REGION Network 4
   RUNG wire#powerrail
      Contact( #Start )
      S_SR(operand := #Automat, r1 := wire#w1)
      S_OFFDT(T_NO := "Spoždění ukončení automatu", TV := S5T#4s, R :=, BI =>, RET_VAL =>)
      Coil( #"Automat Delay" )
   END_RUNG
   RUNG wire#powerrail
      Contact( #Stop )
   END_RUNG wire#w1
   RUNG wire#powerrail
      Contact( "OPPovely"."OP Manual" )
   END_RUNG wire#w1
   // the same network as SCL:
   IF #Start THEN
       #Automat := TRUE;   // SR flip-flop
   END_IF;
   IF #Stop OR "OPPovely"."OP Manual" THEN #Automat := FALSE; END_IF;
   #_s5time1 := S_OFFDT(T_NO := "Spoždění ukončení automatu", S := #Automat, TV := S5T#4s, Q => #_w1);
   #"Automat Delay" := #_w1;
END_REGION

REGION Network 5
   RUNG wire#powerrail
      #"Vyhodnocení hran_Instance"(input := %DB20.DBD0, positive => %DB21.DBD0, negative => %DB22.DBD0)
   END_RUNG
   // the same network as SCL:
   #"Vyhodnocení hran_Instance"(input := %DB20.DBD0, positive => %DB21.DBD0, negative => %DB22.DBD0);   // "Vyhodnocení hran"
END_REGION

REGION Network 6
   RUNG wire#powerrail
      #"Vyhodnocení hran_Instance_Linka 1"(input := %DB20.DBD4, positive => %DB21.DBD4, negative => %DB22.DBD4)
   END_RUNG
   // the same network as SCL:
   #"Vyhodnocení hran_Instance_Linka 1"(input := %DB20.DBD4, positive => %DB21.DBD4, negative => %DB22.DBD4);   // "Vyhodnocení hran"
END_REGION

REGION Network 7
   RUNG wire#powerrail
      Contact( "Tag_64" )
      Coil( "Tag_65" )
   END_RUNG
   // the same network as SCL:
   "Tag_65" := "Tag_64";
END_REGION
END_FUNCTION_BLOCK

FUNCTION_BLOCK "Dopravníky palet_2"   // FB7, LAD
{ S7_Optimized_Access := 'FALSE' }
VERSION : 0.1
   VAR
      Přesun : Struct
         KonecD4naDestohovač : Bool;
         DestohovačNaKonecD5 : Bool;
         KonecD5naZačátekD8 : Bool;
         ZačátekD8naD8pozice12 : Bool;
         D8pozice12naD8pozice11 : Bool;
         D8pozice12naD12 : Bool;
         D8pozice11naD11 : Bool;
         D12naD17pozice12 : Bool;
         D11naD17pozice11 : Bool;
         D17pozice12naKonecP17 : Bool;
         D17pozice11naKonecP17 : Bool;
         KonecP17naZačátekP18 : Bool;
         ZačátekP18naKonecP18 : Bool;
         KonecP18naP19 : Bool;
         P19naZačátekP20 : Bool;
         ZačátekP20naKonecP20 : Bool;
         KonecP20NaP21 : Bool;
      END_STRUCT;
      "Přítomnosti palet" : Struct
         PaletaPodDestohovačem : Bool;
         PaletaNaKonciD5 : Bool;
         PaletaNaZačátkuD8 : Bool;
         PaletaNaD8pozice12 : Bool;
         PaletaNaD8pozice11 : Bool;
         PaletaNaP12 : Bool;
         PaletaNaP11 : Bool;
         PaletaNaD17pozice12 : Bool;
         PaletaNaD17pozice11 : Bool;
         PaletaNaKonciP17 : Bool;
         "PaletaNaZačátku P18" : Bool;
         PaletaNaKonciP18 : Bool;
         PaletaNaP19 : Bool;
         PaletaNaZačátkuP20 : Bool;
         PaletaNaKonciP20 : Bool;
      END_STRUCT;
      "Nájezdy palet" : Struct
         PaletaPodDestohovačem : Bool;
         PaletaNaKonciD5 : Bool;
         PaletaNaZačátkuD8 : Bool;
         PaletaNaD8pozice12 : Bool;
         PaletaNaD8pozice11 : Bool;
         PaletaNaP12 : Bool;
         PaletaNaP11 : Bool;
         PaletaNaD17pozice12 : Bool;
         PaletaNaD17pozice11 : Bool;
         PaletaNaKonciP17 : Bool;
         "PaletaNaZačátku P18" : Bool;
         PaletaNaKonciP18 : Bool;
         PaletaNaP19 : Bool;
         PaletaNaZačátkuP20 : Bool;
         PaletaNaKonciP20 : Bool;
      END_STRUCT;
      Palety : Struct
         P12 : "Paleta";
         P11 : "Paleta";
         P17poziceP11 : "Paleta";
         P17poziceP12 : "Paleta";
         KonecP17 : "Paleta";
         ZačátekP18 : "Paleta";
         KonecP18 : "Paleta";
         P19 : "Paleta";
         ZačátekP20 : "Paleta";
      END_STRUCT;
      Hrany : Struct
         T51Negativní : Bool;
      END_STRUCT;
      "Pallet dispenser_Instance" : "Pallet dispenser";
      "Přítomnost palety_Instance" : "Přítomnost palety";
   END_VAR
   VAR_TEMP
      Dummy : Bool;
      "Rovnání P11 sevřít" : Bool;
      "Rovnání P11 rozevřít" : Bool;
      "Rovnání P12 sevřít" : Bool;
      "Rovnání P12 rozevřít" : Bool;
      "Destohovač sevřít" : Bool;
      "Destohovač rozevřít" : Bool;
   END_VAR
   VAR_TEMP   // added for the SCL form of the ladder/FBD networks
      _s5time1 : S5Time;
      _w1 : Bool;
      _w2 : Bool;
      _w3 : Bool;
   END_VAR
BEGIN

REGION Network 1
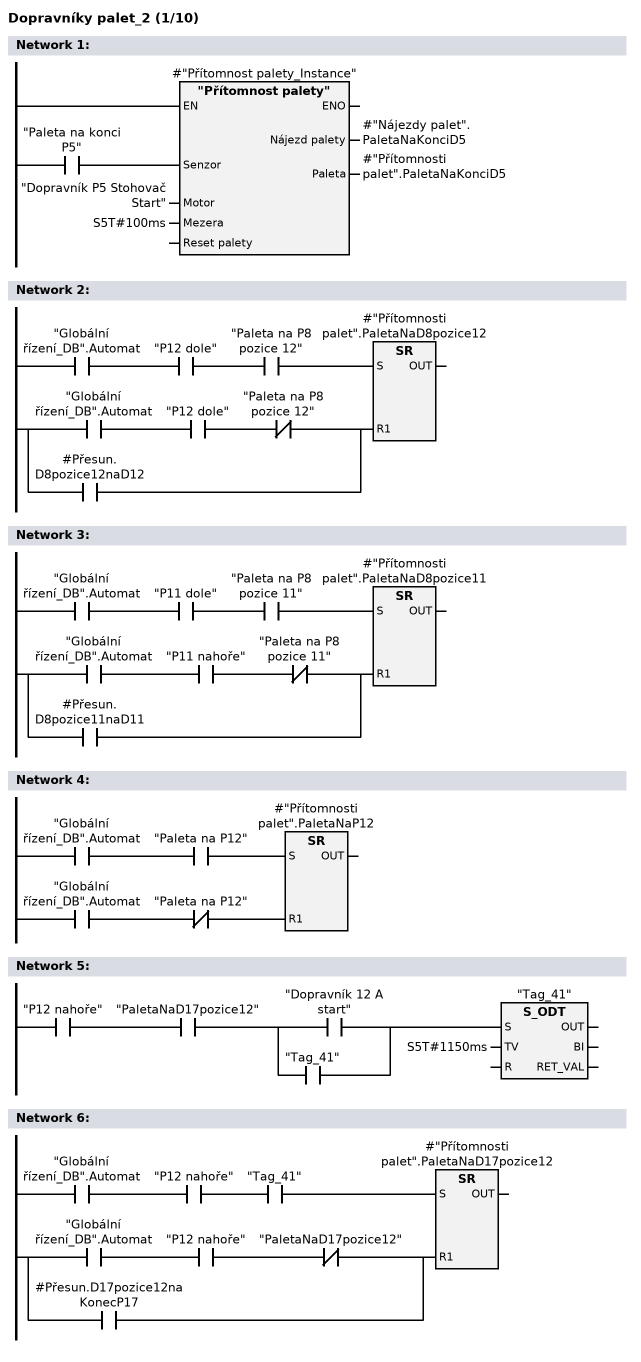
   RUNG wire#powerrail
      #"Přítomnost palety_Instance"(Senzor := wire#w1, Motor := "Dopravník P5 Stohovač Start", Mezera := S5T#100ms, "Reset palety" :=, "Nájezd palety" => #"Nájezdy palet".PaletaNaKonciD5, Paleta => #"Přítomnosti palet".PaletaNaKonciD5)
   END_RUNG
   RUNG wire#powerrail
      Contact( "Paleta na konci P5" )
   END_RUNG wire#w1
   // the same network as SCL:
   #"Přítomnost palety_Instance"(Senzor := "Paleta na konci P5",   // "Přítomnost palety"
                           Motor := "Dopravník P5 Stohovač Start",
                           Mezera := S5T#100ms,
                           "Nájezd palety" => #"Nájezdy palet".PaletaNaKonciD5,
                           Paleta => #"Přítomnosti palet".PaletaNaKonciD5);
END_REGION

REGION Network 2
   RUNG wire#powerrail
      Contact( "Globální řízení_DB".Automat )
      Contact( "P12 dole" )
      Contact( "Paleta na P8 pozice 12" )
      S_SR(operand := #"Přítomnosti palet".PaletaNaD8pozice12, r1 := wire#w1)
   END_RUNG
   RUNG wire#powerrail
      Contact( "Globální řízení_DB".Automat )
      Contact( "P12 dole" )
      I_Contact( "Paleta na P8 pozice 12" )
   END_RUNG wire#w1
   RUNG wire#powerrail
      Contact( #Přesun.D8pozice12naD12 )
   END_RUNG wire#w1
   // the same network as SCL:
   IF "Globální řízení_DB".Automat AND "P12 dole" AND "Paleta na P8 pozice 12" THEN
       #"Přítomnosti palet".PaletaNaD8pozice12 := TRUE;   // SR flip-flop
   END_IF;
   IF ("Globální řízení_DB".Automat AND "P12 dole" AND NOT "Paleta na P8 pozice 12") OR #Přesun.D8pozice12naD12 THEN
       #"Přítomnosti palet".PaletaNaD8pozice12 := FALSE;
   END_IF;
END_REGION

REGION Network 3
   RUNG wire#powerrail
      Contact( "Globální řízení_DB".Automat )
      Contact( "P11 dole" )
      Contact( "Paleta na P8 pozice 11" )
      S_SR(operand := #"Přítomnosti palet".PaletaNaD8pozice11, r1 := wire#w1)
   END_RUNG
   RUNG wire#powerrail
      Contact( "Globální řízení_DB".Automat )
      Contact( "P11 nahoře" )
      I_Contact( "Paleta na P8 pozice 11" )
   END_RUNG wire#w1
   RUNG wire#powerrail
      Contact( #Přesun.D8pozice11naD11 )
   END_RUNG wire#w1
   // the same network as SCL:
   IF "Globální řízení_DB".Automat AND "P11 dole" AND "Paleta na P8 pozice 11" THEN
       #"Přítomnosti palet".PaletaNaD8pozice11 := TRUE;   // SR flip-flop
   END_IF;
   IF ("Globální řízení_DB".Automat AND "P11 nahoře" AND NOT "Paleta na P8 pozice 11") OR #Přesun.D8pozice11naD11 THEN
       #"Přítomnosti palet".PaletaNaD8pozice11 := FALSE;
   END_IF;
END_REGION

REGION Network 4
   RUNG wire#powerrail
      Contact( "Globální řízení_DB".Automat )
      Contact( "Paleta na P12" )
      S_SR(operand := #"Přítomnosti palet".PaletaNaP12, r1 := wire#w1)
   END_RUNG
   RUNG wire#powerrail
      Contact( "Globální řízení_DB".Automat )
      I_Contact( "Paleta na P12" )
   END_RUNG wire#w1
   // the same network as SCL:
   IF "Globální řízení_DB".Automat AND "Paleta na P12" THEN
       #"Přítomnosti palet".PaletaNaP12 := TRUE;   // SR flip-flop
   END_IF;
   IF "Globální řízení_DB".Automat AND NOT "Paleta na P12" THEN
       #"Přítomnosti palet".PaletaNaP12 := FALSE;
   END_IF;
END_REGION

REGION Network 5
   RUNG wire#powerrail
      Contact( "P12 nahoře" )
      Contact( "PaletaNaD17pozice12" )
      wire#w1
      Contact( "Dopravník 12 A start" )
      wire#w2
      S_ODT(T_NO := "Tag_41", TV := S5T#1150ms, R :=, BI =>, RET_VAL =>)
   END_RUNG
   RUNG wire#w1
      Contact( "Tag_41" )
   END_RUNG wire#w2
   // the same network as SCL:
   #_s5time1 := S_ODT(T_NO := "Tag_41",
                      S := "P12 nahoře" AND "PaletaNaD17pozice12" AND ("Dopravník 12 A start" OR "Tag_41"),
                      TV := S5T#1150ms);
END_REGION

REGION Network 6
   RUNG wire#powerrail
      Contact( "Globální řízení_DB".Automat )
      Contact( "P12 nahoře" )
      Contact( "Tag_41" )
      S_SR(operand := #"Přítomnosti palet".PaletaNaD17pozice12, r1 := wire#w1)
   END_RUNG
   RUNG wire#powerrail
      Contact( "Globální řízení_DB".Automat )
      Contact( "P12 nahoře" )
      I_Contact( "PaletaNaD17pozice12" )
   END_RUNG wire#w1
   RUNG wire#powerrail
      Contact( #Přesun.D17pozice12naKonecP17 )
   END_RUNG wire#w1
   // the same network as SCL:
   IF "Globální řízení_DB".Automat AND "P12 nahoře" AND "Tag_41" THEN
       #"Přítomnosti palet".PaletaNaD17pozice12 := TRUE;   // SR flip-flop
   END_IF;
   IF ("Globální řízení_DB".Automat AND "P12 nahoře" AND NOT "PaletaNaD17pozice12") OR #Přesun.D17pozice12naKonecP17 THEN
       #"Přítomnosti palet".PaletaNaD17pozice12 := FALSE;
   END_IF;
END_REGION

REGION Network 7
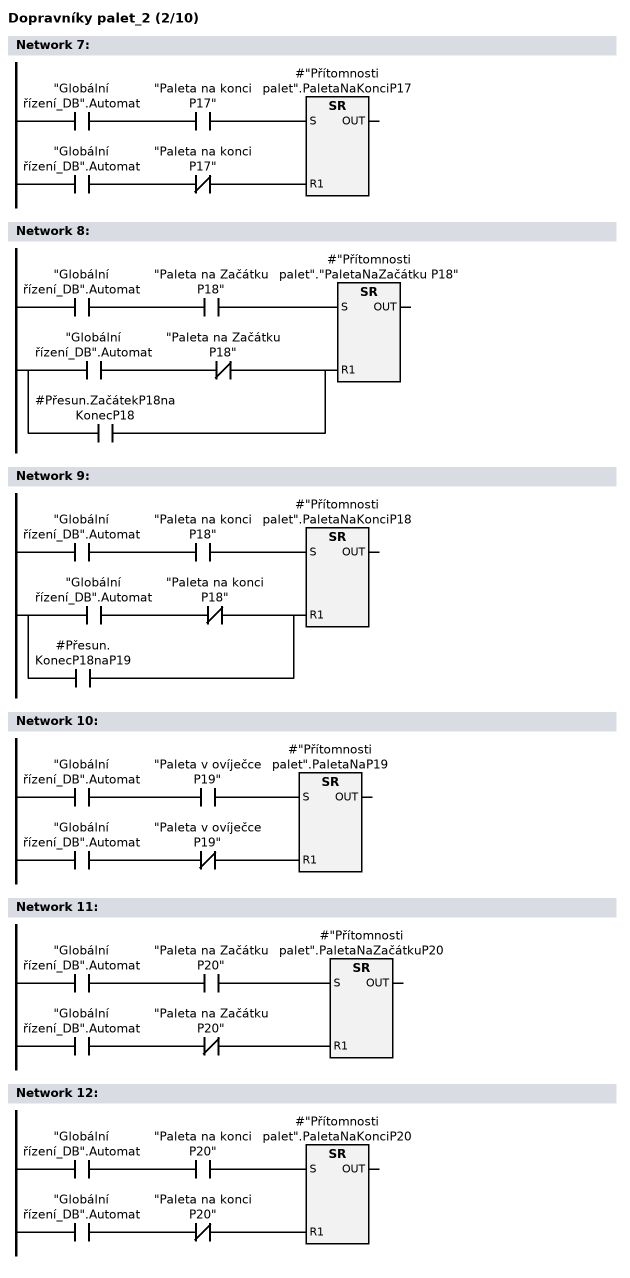
   RUNG wire#powerrail
      Contact( "Globální řízení_DB".Automat )
      Contact( "Paleta na konci P17" )
      S_SR(operand := #"Přítomnosti palet".PaletaNaKonciP17, r1 := wire#w1)
   END_RUNG
   RUNG wire#powerrail
      Contact( "Globální řízení_DB".Automat )
      I_Contact( "Paleta na konci P17" )
   END_RUNG wire#w1
   // the same network as SCL:
   IF "Globální řízení_DB".Automat AND "Paleta na konci P17" THEN
       #"Přítomnosti palet".PaletaNaKonciP17 := TRUE;   // SR flip-flop
   END_IF;
   IF "Globální řízení_DB".Automat AND NOT "Paleta na konci P17" THEN
       #"Přítomnosti palet".PaletaNaKonciP17 := FALSE;
   END_IF;
END_REGION

REGION Network 8
   RUNG wire#powerrail
      Contact( "Globální řízení_DB".Automat )
      Contact( "Paleta na Začátku P18" )
      S_SR(operand := #"Přítomnosti palet"."PaletaNaZačátku P18", r1 := wire#w1)
   END_RUNG
   RUNG wire#powerrail
      Contact( "Globální řízení_DB".Automat )
      I_Contact( "Paleta na Začátku P18" )
   END_RUNG wire#w1
   RUNG wire#powerrail
      Contact( #Přesun.ZačátekP18naKonecP18 )
   END_RUNG wire#w1
   // the same network as SCL:
   IF "Globální řízení_DB".Automat AND "Paleta na Začátku P18" THEN
       #"Přítomnosti palet"."PaletaNaZačátku P18" := TRUE;   // SR flip-flop
   END_IF;
   IF ("Globální řízení_DB".Automat AND NOT "Paleta na Začátku P18") OR #Přesun.ZačátekP18naKonecP18 THEN
       #"Přítomnosti palet"."PaletaNaZačátku P18" := FALSE;
   END_IF;
END_REGION

REGION Network 9
   RUNG wire#powerrail
      Contact( "Globální řízení_DB".Automat )
      Contact( "Paleta na konci P18" )
      S_SR(operand := #"Přítomnosti palet".PaletaNaKonciP18, r1 := wire#w1)
   END_RUNG
   RUNG wire#powerrail
      Contact( "Globální řízení_DB".Automat )
      I_Contact( "Paleta na konci P18" )
   END_RUNG wire#w1
   RUNG wire#powerrail
      Contact( #Přesun.KonecP18naP19 )
   END_RUNG wire#w1
   // the same network as SCL:
   IF "Globální řízení_DB".Automat AND "Paleta na konci P18" THEN
       #"Přítomnosti palet".PaletaNaKonciP18 := TRUE;   // SR flip-flop
   END_IF;
   IF ("Globální řízení_DB".Automat AND NOT "Paleta na konci P18") OR #Přesun.KonecP18naP19 THEN
       #"Přítomnosti palet".PaletaNaKonciP18 := FALSE;
   END_IF;
END_REGION

REGION Network 10
   RUNG wire#powerrail
      Contact( "Globální řízení_DB".Automat )
      Contact( "Paleta v ovíječce P19" )
      S_SR(operand := #"Přítomnosti palet".PaletaNaP19, r1 := wire#w1)
   END_RUNG
   RUNG wire#powerrail
      Contact( "Globální řízení_DB".Automat )
      I_Contact( "Paleta v ovíječce P19" )
   END_RUNG wire#w1
   // the same network as SCL:
   IF "Globální řízení_DB".Automat AND "Paleta v ovíječce P19" THEN
       #"Přítomnosti palet".PaletaNaP19 := TRUE;   // SR flip-flop
   END_IF;
   IF "Globální řízení_DB".Automat AND NOT "Paleta v ovíječce P19" THEN
       #"Přítomnosti palet".PaletaNaP19 := FALSE;
   END_IF;
END_REGION

REGION Network 11
   RUNG wire#powerrail
      Contact( "Globální řízení_DB".Automat )
      Contact( "Paleta na Začátku P20" )
      S_SR(operand := #"Přítomnosti palet".PaletaNaZačátkuP20, r1 := wire#w1)
   END_RUNG
   RUNG wire#powerrail
      Contact( "Globální řízení_DB".Automat )
      I_Contact( "Paleta na Začátku P20" )
   END_RUNG wire#w1
   // the same network as SCL:
   IF "Globální řízení_DB".Automat AND "Paleta na Začátku P20" THEN
       #"Přítomnosti palet".PaletaNaZačátkuP20 := TRUE;   // SR flip-flop
   END_IF;
   IF "Globální řízení_DB".Automat AND NOT "Paleta na Začátku P20" THEN
       #"Přítomnosti palet".PaletaNaZačátkuP20 := FALSE;
   END_IF;
END_REGION

REGION Network 12
   RUNG wire#powerrail
      Contact( "Globální řízení_DB".Automat )
      Contact( "Paleta na konci P20" )
      S_SR(operand := #"Přítomnosti palet".PaletaNaKonciP20, r1 := wire#w1)
   END_RUNG
   RUNG wire#powerrail
      Contact( "Globální řízení_DB".Automat )
      I_Contact( "Paleta na konci P20" )
   END_RUNG wire#w1
   // the same network as SCL:
   IF "Globální řízení_DB".Automat AND "Paleta na konci P20" THEN
       #"Přítomnosti palet".PaletaNaKonciP20 := TRUE;   // SR flip-flop
   END_IF;
   IF "Globální řízení_DB".Automat AND NOT "Paleta na konci P20" THEN
       #"Přítomnosti palet".PaletaNaKonciP20 := FALSE;
   END_IF;
END_REGION

REGION Network 13
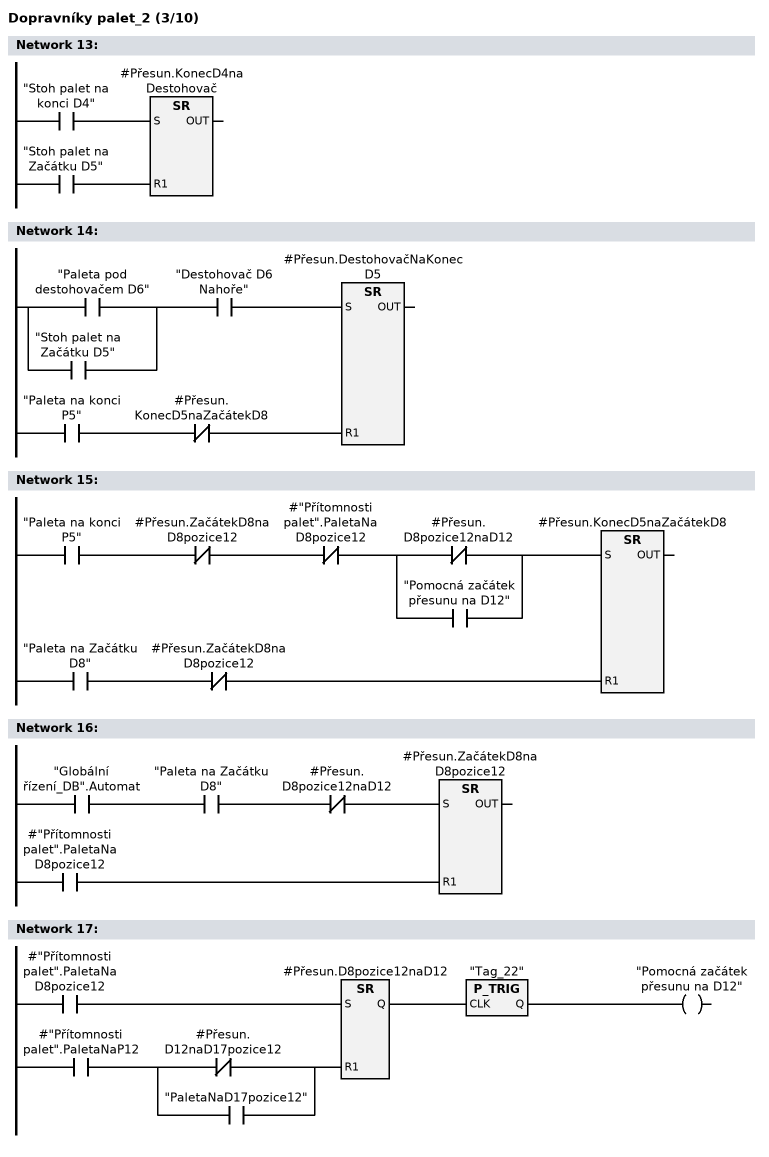
   RUNG wire#powerrail
      Contact( "Stoh palet na konci D4" )
      S_SR(operand := #Přesun.KonecD4naDestohovač, r1 := wire#w1)
   END_RUNG
   RUNG wire#powerrail
      Contact( "Stoh palet na Začátku D5" )
   END_RUNG wire#w1
   // the same network as SCL:
   IF "Stoh palet na konci D4" THEN
       #Přesun.KonecD4naDestohovač := TRUE;   // SR flip-flop
   END_IF;
   IF "Stoh palet na Začátku D5" THEN #Přesun.KonecD4naDestohovač := FALSE; END_IF;
END_REGION

REGION Network 14
   RUNG wire#powerrail
      Contact( "Paleta pod destohovačem D6" )
      wire#w1
      Contact( "Destohovač D6 Nahoře" )
      S_SR(operand := #Přesun.DestohovačNaKonecD5, r1 := wire#w2)
   END_RUNG
   RUNG wire#powerrail
      Contact( "Stoh palet na Začátku D5" )
   END_RUNG wire#w1
   RUNG wire#powerrail
      Contact( "Paleta na konci P5" )
      I_Contact( #Přesun.KonecD5naZačátekD8 )
   END_RUNG wire#w2
   // the same network as SCL:
   IF ("Paleta pod destohovačem D6" OR "Stoh palet na Začátku D5") AND "Destohovač D6 Nahoře" THEN
       #Přesun.DestohovačNaKonecD5 := TRUE;   // SR flip-flop
   END_IF;
   IF "Paleta na konci P5" AND NOT #Přesun.KonecD5naZačátekD8 THEN
       #Přesun.DestohovačNaKonecD5 := FALSE;
   END_IF;
END_REGION

REGION Network 15
   RUNG wire#powerrail
      Contact( "Paleta na konci P5" )
      I_Contact( #Přesun.ZačátekD8naD8pozice12 )
      I_Contact( #"Přítomnosti palet".PaletaNaD8pozice12 )
      wire#w1
      I_Contact( #Přesun.D8pozice12naD12 )
      wire#w2
      S_SR(operand := #Přesun.KonecD5naZačátekD8, r1 := wire#w3)
   END_RUNG
   RUNG wire#w1
      Contact( "Pomocná začátek přesunu na D12" )
   END_RUNG wire#w2
   RUNG wire#powerrail
      Contact( "Paleta na Začátku D8" )
      I_Contact( #Přesun.ZačátekD8naD8pozice12 )
   END_RUNG wire#w3
   // the same network as SCL:
   IF "Paleta na konci P5" AND NOT #Přesun.ZačátekD8naD8pozice12 AND NOT #"Přítomnosti palet".PaletaNaD8pozice12 AND (NOT #Přesun.D8pozice12naD12 OR "Pomocná začátek přesunu na D12") THEN
       #Přesun.KonecD5naZačátekD8 := TRUE;   // SR flip-flop
   END_IF;
   IF "Paleta na Začátku D8" AND NOT #Přesun.ZačátekD8naD8pozice12 THEN
       #Přesun.KonecD5naZačátekD8 := FALSE;
   END_IF;
END_REGION

REGION Network 16
   RUNG wire#powerrail
      Contact( "Globální řízení_DB".Automat )
      Contact( "Paleta na Začátku D8" )
      I_Contact( #Přesun.D8pozice12naD12 )
      S_SR(operand := #Přesun.ZačátekD8naD8pozice12, r1 := wire#w1)
   END_RUNG
   RUNG wire#powerrail
      Contact( #"Přítomnosti palet".PaletaNaD8pozice12 )
   END_RUNG wire#w1
   // the same network as SCL:
   IF "Globální řízení_DB".Automat AND "Paleta na Začátku D8" AND NOT #Přesun.D8pozice12naD12 THEN
       #Přesun.ZačátekD8naD8pozice12 := TRUE;   // SR flip-flop
   END_IF;
   IF #"Přítomnosti palet".PaletaNaD8pozice12 THEN #Přesun.ZačátekD8naD8pozice12 := FALSE; END_IF;
END_REGION

REGION Network 17
   RUNG wire#powerrail
      Contact( #"Přítomnosti palet".PaletaNaD8pozice12 )
      S_SR(operand := #Přesun.D8pozice12naD12, r1 := wire#w2)
      P_Trig( "Tag_22" )
      Coil( "Pomocná začátek přesunu na D12" )
   END_RUNG
   RUNG wire#powerrail
      Contact( #"Přítomnosti palet".PaletaNaP12 )
      wire#w1
      I_Contact( #Přesun.D12naD17pozice12 )
   END_RUNG wire#w2
   RUNG wire#w1
      Contact( "PaletaNaD17pozice12" )
   END_RUNG wire#w2
   // the same network as SCL:
   IF #"Přítomnosti palet".PaletaNaD8pozice12 THEN
       #Přesun.D8pozice12naD12 := TRUE;   // SR flip-flop
   END_IF;
   IF #"Přítomnosti palet".PaletaNaP12 AND (NOT #Přesun.D12naD17pozice12 OR "PaletaNaD17pozice12") THEN
       #Přesun.D8pozice12naD12 := FALSE;
   END_IF;
   #_w1 := #Přesun.D8pozice12naD12 AND NOT "Tag_22";   // rising edge
   "Tag_22" := #Přesun.D8pozice12naD12;
   "Pomocná začátek přesunu na D12" := #_w1;
END_REGION

REGION Network 18
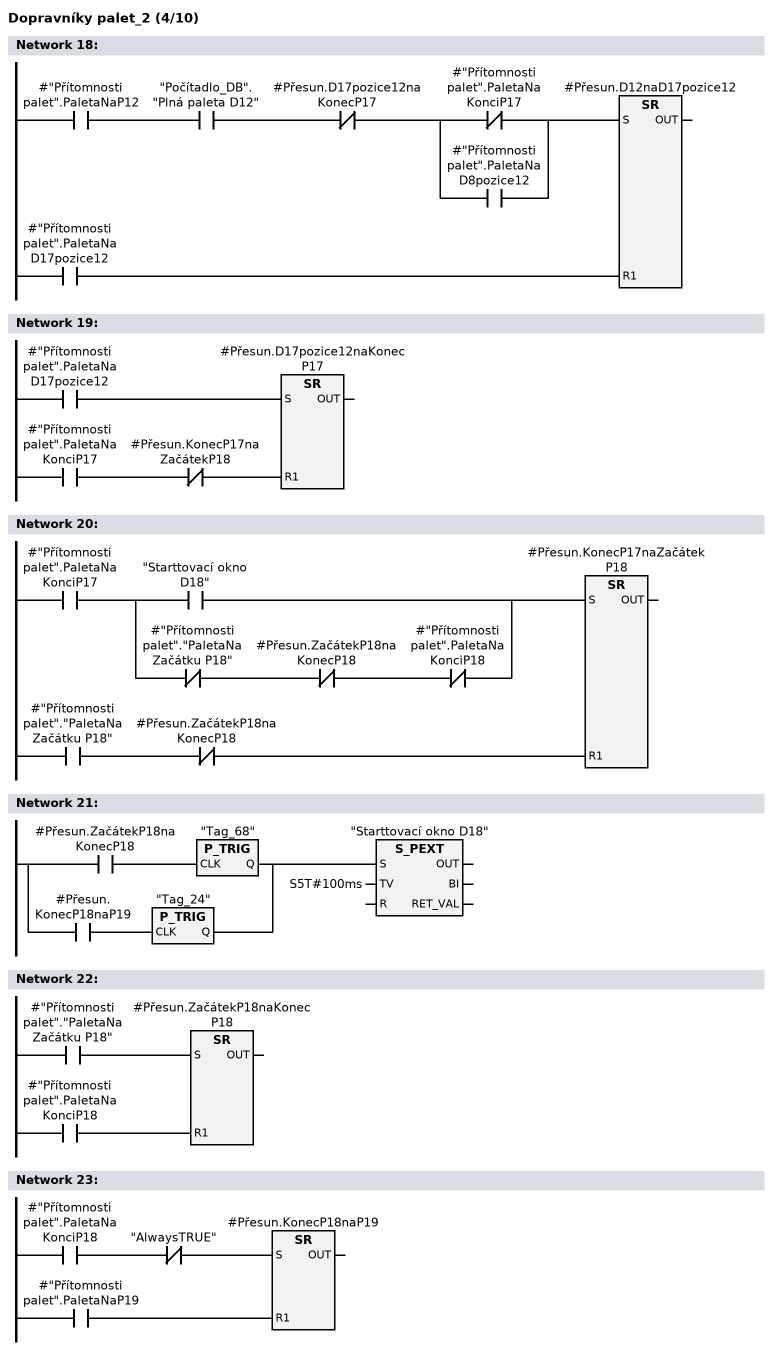
   RUNG wire#powerrail
      Contact( #"Přítomnosti palet".PaletaNaP12 )
      Contact( "Počítadlo_DB"."Plná paleta D12" )
      I_Contact( #Přesun.D17pozice12naKonecP17 )
      wire#w1
      I_Contact( #"Přítomnosti palet".PaletaNaKonciP17 )
      wire#w2
      S_SR(operand := #Přesun.D12naD17pozice12, r1 := wire#w3)
   END_RUNG
   RUNG wire#w1
      Contact( #"Přítomnosti palet".PaletaNaD8pozice12 )
   END_RUNG wire#w2
   RUNG wire#powerrail
      Contact( #"Přítomnosti palet".PaletaNaD17pozice12 )
   END_RUNG wire#w3
   // the same network as SCL:
   IF #"Přítomnosti palet".PaletaNaP12 AND "Počítadlo_DB"."Plná paleta D12" AND NOT #Přesun.D17pozice12naKonecP17 AND (NOT #"Přítomnosti palet".PaletaNaKonciP17 OR #"Přítomnosti palet".PaletaNaD8pozice12) THEN
       #Přesun.D12naD17pozice12 := TRUE;   // SR flip-flop
   END_IF;
   IF #"Přítomnosti palet".PaletaNaD17pozice12 THEN #Přesun.D12naD17pozice12 := FALSE; END_IF;
END_REGION

REGION Network 19
   RUNG wire#powerrail
      Contact( #"Přítomnosti palet".PaletaNaD17pozice12 )
      S_SR(operand := #Přesun.D17pozice12naKonecP17, r1 := wire#w1)
   END_RUNG
   RUNG wire#powerrail
      Contact( #"Přítomnosti palet".PaletaNaKonciP17 )
      I_Contact( #Přesun.KonecP17naZačátekP18 )
   END_RUNG wire#w1
   // the same network as SCL:
   IF #"Přítomnosti palet".PaletaNaD17pozice12 THEN
       #Přesun.D17pozice12naKonecP17 := TRUE;   // SR flip-flop
   END_IF;
   IF #"Přítomnosti palet".PaletaNaKonciP17 AND NOT #Přesun.KonecP17naZačátekP18 THEN
       #Přesun.D17pozice12naKonecP17 := FALSE;
   END_IF;
END_REGION

REGION Network 20
   RUNG wire#powerrail
      Contact( #"Přítomnosti palet".PaletaNaKonciP17 )
      wire#w1
      Contact( "Starttovací okno D18" )
      wire#w2
      S_SR(operand := #Přesun.KonecP17naZačátekP18, r1 := wire#w3)
   END_RUNG
   RUNG wire#w1
      I_Contact( #"Přítomnosti palet"."PaletaNaZačátku P18" )
      I_Contact( #Přesun.ZačátekP18naKonecP18 )
      I_Contact( #"Přítomnosti palet".PaletaNaKonciP18 )
   END_RUNG wire#w2
   RUNG wire#powerrail
      Contact( #"Přítomnosti palet"."PaletaNaZačátku P18" )
      I_Contact( #Přesun.ZačátekP18naKonecP18 )
   END_RUNG wire#w3
   // the same network as SCL:
   IF #"Přítomnosti palet".PaletaNaKonciP17 AND ("Starttovací okno D18" OR (NOT #"Přítomnosti palet"."PaletaNaZačátku P18" AND NOT #Přesun.ZačátekP18naKonecP18 AND NOT #"Přítomnosti palet".PaletaNaKonciP18)) THEN
       #Přesun.KonecP17naZačátekP18 := TRUE;   // SR flip-flop
   END_IF;
   IF #"Přítomnosti palet"."PaletaNaZačátku P18" AND NOT #Přesun.ZačátekP18naKonecP18 THEN
       #Přesun.KonecP17naZačátekP18 := FALSE;
   END_IF;
END_REGION

REGION Network 21
   RUNG wire#powerrail
      Contact( #Přesun.ZačátekP18naKonecP18 )
      P_Trig( "Tag_68" )
      wire#w1
      S_PEXT(T_NO := "Starttovací okno D18", TV := S5T#100ms, R :=, BI =>, RET_VAL =>)
   END_RUNG
   RUNG wire#powerrail
      Contact( #Přesun.KonecP18naP19 )
      P_Trig( "Tag_24" )
   END_RUNG wire#w1
   // the same network as SCL:
   #_w1 := #Přesun.ZačátekP18naKonecP18 AND NOT "Tag_68";   // rising edge
   "Tag_68" := #Přesun.ZačátekP18naKonecP18;
   #_w2 := #Přesun.KonecP18naP19 AND NOT "Tag_24";   // rising edge
   "Tag_24" := #Přesun.KonecP18naP19;
   #_s5time1 := S_PEXT(T_NO := "Starttovací okno D18", S := #_w1 OR #_w2, TV := S5T#100ms);
END_REGION

REGION Network 22
   RUNG wire#powerrail
      Contact( #"Přítomnosti palet"."PaletaNaZačátku P18" )
      S_SR(operand := #Přesun.ZačátekP18naKonecP18, r1 := wire#w1)
   END_RUNG
   RUNG wire#powerrail
      Contact( #"Přítomnosti palet".PaletaNaKonciP18 )
   END_RUNG wire#w1
   // the same network as SCL:
   IF #"Přítomnosti palet"."PaletaNaZačátku P18" THEN
       #Přesun.ZačátekP18naKonecP18 := TRUE;   // SR flip-flop
   END_IF;
   IF #"Přítomnosti palet".PaletaNaKonciP18 THEN #Přesun.ZačátekP18naKonecP18 := FALSE; END_IF;
END_REGION

REGION Network 23
   RUNG wire#powerrail
      Contact( #"Přítomnosti palet".PaletaNaKonciP18 )
      I_Contact( "AlwaysTRUE" )
      S_SR(operand := #Přesun.KonecP18naP19, r1 := wire#w1)
   END_RUNG
   RUNG wire#powerrail
      Contact( #"Přítomnosti palet".PaletaNaP19 )
   END_RUNG wire#w1
   // the same network as SCL:
   IF #"Přítomnosti palet".PaletaNaKonciP18 AND NOT "AlwaysTRUE" THEN
       #Přesun.KonecP18naP19 := TRUE;   // SR flip-flop
   END_IF;
   IF #"Přítomnosti palet".PaletaNaP19 THEN #Přesun.KonecP18naP19 := FALSE; END_IF;
END_REGION

REGION Network 24
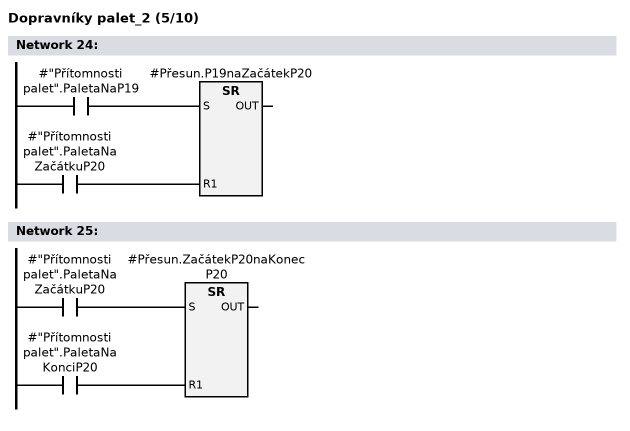
   RUNG wire#powerrail
      Contact( #"Přítomnosti palet".PaletaNaP19 )
      S_SR(operand := #Přesun.P19naZačátekP20, r1 := wire#w1)
   END_RUNG
   RUNG wire#powerrail
      Contact( #"Přítomnosti palet".PaletaNaZačátkuP20 )
   END_RUNG wire#w1
   // the same network as SCL:
   IF #"Přítomnosti palet".PaletaNaP19 THEN
       #Přesun.P19naZačátekP20 := TRUE;   // SR flip-flop
   END_IF;
   IF #"Přítomnosti palet".PaletaNaZačátkuP20 THEN #Přesun.P19naZačátekP20 := FALSE; END_IF;
END_REGION

REGION Network 25
   RUNG wire#powerrail
      Contact( #"Přítomnosti palet".PaletaNaZačátkuP20 )
      S_SR(operand := #Přesun.ZačátekP20naKonecP20, r1 := wire#w1)
   END_RUNG
   RUNG wire#powerrail
      Contact( #"Přítomnosti palet".PaletaNaKonciP20 )
   END_RUNG wire#w1
   // the same network as SCL:
   IF #"Přítomnosti palet".PaletaNaZačátkuP20 THEN
       #Přesun.ZačátekP20naKonecP20 := TRUE;   // SR flip-flop
   END_IF;
   IF #"Přítomnosti palet".PaletaNaKonciP20 THEN #Přesun.ZačátekP20naKonecP20 := FALSE; END_IF;
END_REGION

REGION Network 26
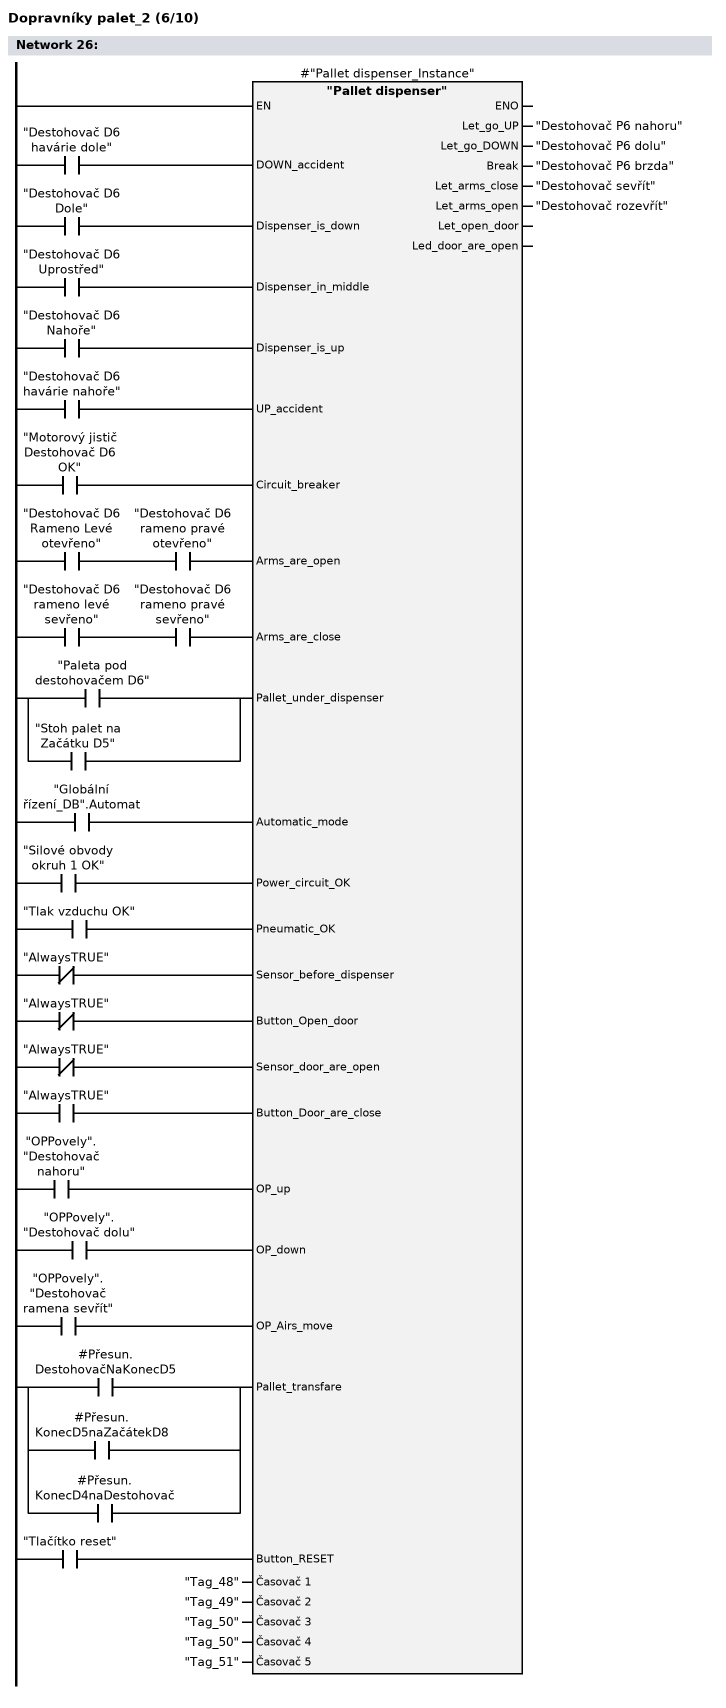
   RUNG wire#powerrail
      #"Pallet dispenser_Instance"(DOWN_accident := wire#w1, Dispenser_is_down := wire#w2, Dispenser_in_middle := wire#w3, Dispenser_is_up := wire#w4, UP_accident := wire#w5, Circuit_breaker := wire#w6, Arms_are_open := wire#w7, Arms_are_close := wire#w8, Pallet_under_dispenser := wire#w9, Automatic_mode := wire#w10, Power_circuit_OK := wire#w11, Pneumatic_OK := wire#w12, Sensor_before_dispenser := wire#w13, Button_Open_door := wire#w14, Sensor_door_are_open := wire#w15, Button_Door_are_close := wire#w16, OP_up := wire#w17, OP_down := wire#w18, OP_Airs_move := wire#w19, Pallet_transfare := wire#w20, Button_RESET := wire#w21, "Časovač 1" := "Tag_48", "Časovač 2" := "Tag_49", "Časovač 3" := "Tag_50", "Časovač 4" := "Tag_50", "Časovač 5" := "Tag_51", Let_go_UP => "Destohovač P6 nahoru", Let_go_DOWN => "Destohovač P6 dolu", Break => "Destohovač P6 brzda", Let_arms_close => "Destohovač sevřít", Let_arms_open => "Destohovač rozevřít", Let_open_door =>, Led_door_are_open =>)
   END_RUNG
   RUNG wire#powerrail
      Contact( "Destohovač D6 havárie dole" )
   END_RUNG wire#w1
   RUNG wire#powerrail
      Contact( "Destohovač D6 Dole" )
   END_RUNG wire#w2
   RUNG wire#powerrail
      Contact( "Destohovač D6 Uprostřed" )
   END_RUNG wire#w3
   RUNG wire#powerrail
      Contact( "Destohovač D6 Nahoře" )
   END_RUNG wire#w4
   RUNG wire#powerrail
      Contact( "Destohovač D6 havárie nahoře" )
   END_RUNG wire#w5
   RUNG wire#powerrail
      Contact( "Motorový jistič Destohovač D6 OK" )
   END_RUNG wire#w6
   RUNG wire#powerrail
      Contact( "Destohovač D6 Rameno Levé otevřeno" )
      Contact( "Destohovač D6 rameno pravé otevřeno" )
   END_RUNG wire#w7
   RUNG wire#powerrail
      Contact( "Destohovač D6 rameno levé sevřeno" )
      Contact( "Destohovač D6 rameno pravé sevřeno" )
   END_RUNG wire#w8
   RUNG wire#powerrail
      Contact( "Paleta pod destohovačem D6" )
   END_RUNG wire#w9
   RUNG wire#powerrail
      Contact( "Stoh palet na Začátku D5" )
   END_RUNG wire#w9
   RUNG wire#powerrail
      Contact( "Globální řízení_DB".Automat )
   END_RUNG wire#w10
   RUNG wire#powerrail
      Contact( "Silové obvody okruh 1 OK" )
   END_RUNG wire#w11
   RUNG wire#powerrail
      Contact( "Tlak vzduchu OK" )
   END_RUNG wire#w12
   RUNG wire#powerrail
      I_Contact( "AlwaysTRUE" )
   END_RUNG wire#w13
   RUNG wire#powerrail
      I_Contact( "AlwaysTRUE" )
   END_RUNG wire#w14
   RUNG wire#powerrail
      I_Contact( "AlwaysTRUE" )
   END_RUNG wire#w15
   RUNG wire#powerrail
      Contact( "AlwaysTRUE" )
   END_RUNG wire#w16
   RUNG wire#powerrail
      Contact( "OPPovely"."Destohovač nahoru" )
   END_RUNG wire#w17
   RUNG wire#powerrail
      Contact( "OPPovely"."Destohovač dolu" )
   END_RUNG wire#w18
   RUNG wire#powerrail
      Contact( "OPPovely"."Destohovač ramena sevřít" )
   END_RUNG wire#w19
   RUNG wire#powerrail
      Contact( #Přesun.DestohovačNaKonecD5 )
   END_RUNG wire#w20
   RUNG wire#powerrail
      Contact( #Přesun.KonecD5naZačátekD8 )
   END_RUNG wire#w20
   RUNG wire#powerrail
      Contact( #Přesun.KonecD4naDestohovač )
   END_RUNG wire#w20
   RUNG wire#powerrail
      Contact( "Tlačítko reset" )
   END_RUNG wire#w21
   // the same network as SCL:
   #"Pallet dispenser_Instance"(DOWN_accident := "Destohovač D6 havárie dole",   // "Pallet dispenser"
                           Dispenser_is_down := "Destohovač D6 Dole",
                           Dispenser_in_middle := "Destohovač D6 Uprostřed",
                           Dispenser_is_up := "Destohovač D6 Nahoře",
                           UP_accident := "Destohovač D6 havárie nahoře",
                           Circuit_breaker := "Motorový jistič Destohovač D6 OK",
                           Arms_are_open := "Destohovač D6 Rameno Levé otevřeno" AND "Destohovač D6 rameno pravé otevřeno",
                           Arms_are_close := "Destohovač D6 rameno levé sevřeno" AND "Destohovač D6 rameno pravé sevřeno",
                           Pallet_under_dispenser := "Paleta pod destohovačem D6" OR "Stoh palet na Začátku D5",
                           Automatic_mode := "Globální řízení_DB".Automat,
                           Power_circuit_OK := "Silové obvody okruh 1 OK",
                           Pneumatic_OK := "Tlak vzduchu OK",
                           Sensor_before_dispenser := NOT "AlwaysTRUE",
                           Button_Open_door := NOT "AlwaysTRUE",
                           Sensor_door_are_open := NOT "AlwaysTRUE",
                           Button_Door_are_close := "AlwaysTRUE",
                           OP_up := "OPPovely"."Destohovač nahoru",
                           OP_down := "OPPovely"."Destohovač dolu",
                           OP_Airs_move := "OPPovely"."Destohovač ramena sevřít",
                           Pallet_transfare := #Přesun.DestohovačNaKonecD5 OR #Přesun.KonecD5naZačátekD8 OR #Přesun.KonecD4naDestohovač,
                           Button_RESET := "Tlačítko reset",
                           "Časovač 1" := "Tag_48",
                           "Časovač 2" := "Tag_49",
                           "Časovač 3" := "Tag_50",
                           "Časovač 4" := "Tag_50",
                           "Časovač 5" := "Tag_51",
                           Let_go_UP => "Destohovač P6 nahoru",
                           Let_go_DOWN => "Destohovač P6 dolu",
                           Break => "Destohovač P6 brzda",
                           Let_arms_close => "Destohovač sevřít",
                           Let_arms_open => "Destohovač rozevřít");
END_REGION

REGION Network 27
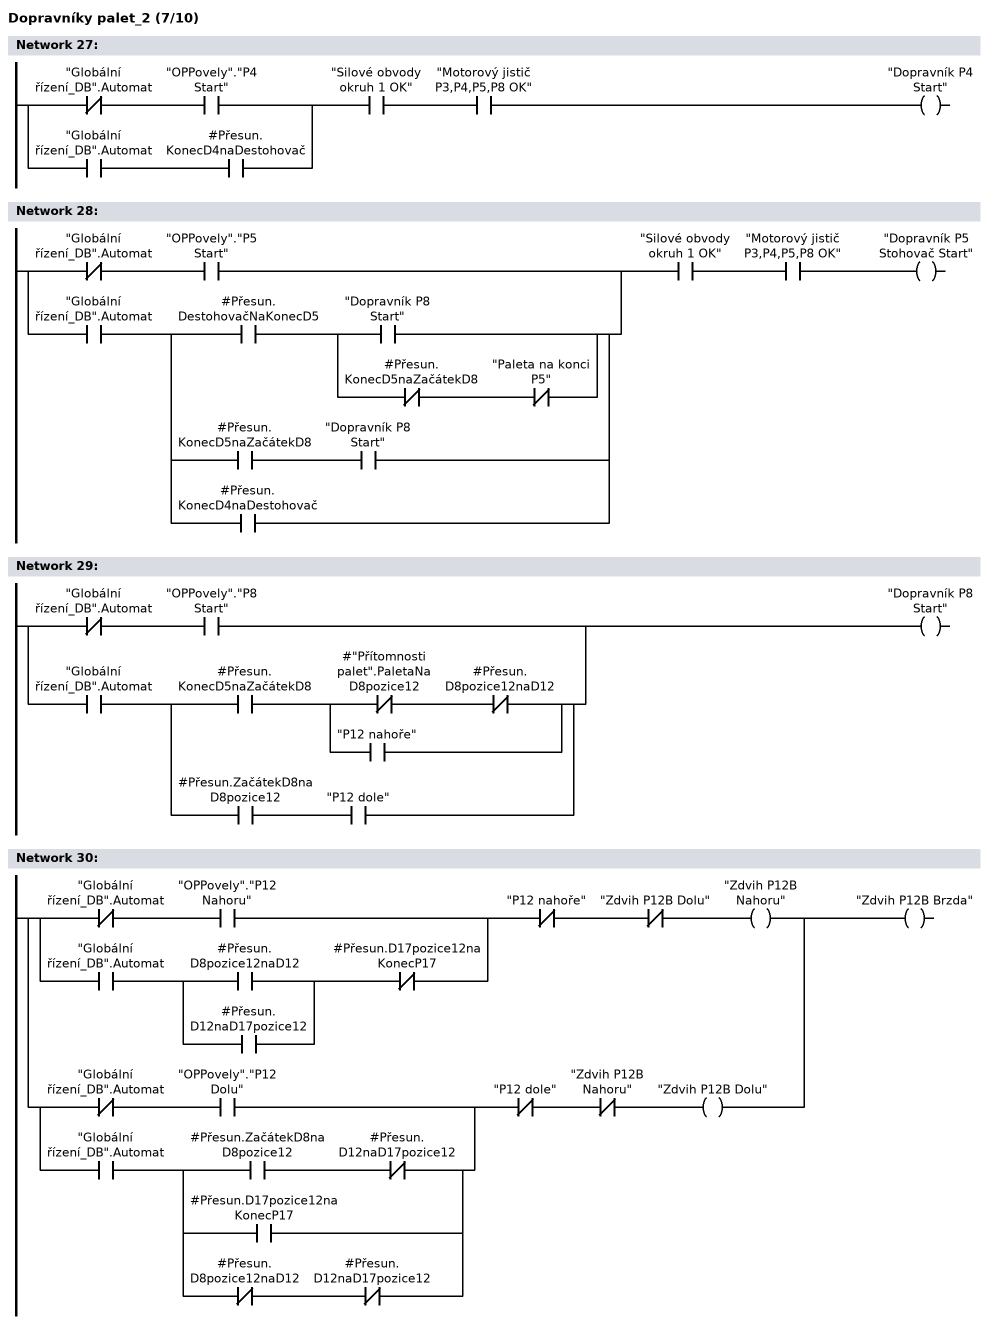
   RUNG wire#powerrail
      I_Contact( "Globální řízení_DB".Automat )
      Contact( "OPPovely"."P4 Start" )
      wire#w1
      Contact( "Silové obvody okruh 1 OK" )
      Contact( "Motorový jistič P3,P4,P5,P8 OK" )
      Coil( "Dopravník P4 Start" )
   END_RUNG
   RUNG wire#powerrail
      Contact( "Globální řízení_DB".Automat )
      Contact( #Přesun.KonecD4naDestohovač )
   END_RUNG wire#w1
   // the same network as SCL:
   "Dopravník P4 Start" := ((NOT "Globální řízení_DB".Automat AND "OPPovely"."P4 Start") OR ("Globální řízení_DB".Automat AND #Přesun.KonecD4naDestohovač)) AND "Silové obvody okruh 1 OK" AND "Motorový jistič P3,P4,P5,P8 OK";
END_REGION

REGION Network 28
   RUNG wire#powerrail
      I_Contact( "Globální řízení_DB".Automat )
      Contact( "OPPovely"."P5 Start" )
      wire#w1
      Contact( "Silové obvody okruh 1 OK" )
      Contact( "Motorový jistič P3,P4,P5,P8 OK" )
      Coil( "Dopravník P5 Stohovač Start" )
   END_RUNG
   RUNG wire#powerrail
      Contact( "Globální řízení_DB".Automat )
      wire#w2
      Contact( #Přesun.DestohovačNaKonecD5 )
      wire#w3
      Contact( "Dopravník P8 Start" )
   END_RUNG wire#w1
   RUNG wire#w3
      I_Contact( #Přesun.KonecD5naZačátekD8 )
      I_Contact( "Paleta na konci P5" )
   END_RUNG wire#w1
   RUNG wire#w2
      Contact( #Přesun.KonecD5naZačátekD8 )
      Contact( "Dopravník P8 Start" )
   END_RUNG wire#w1
   RUNG wire#w2
      Contact( #Přesun.KonecD4naDestohovač )
   END_RUNG wire#w1
   // the same network as SCL:
   "Dopravník P5 Stohovač Start" := ((NOT "Globální řízení_DB".Automat AND "OPPovely"."P5 Start") OR ("Globální řízení_DB".Automat AND ((#Přesun.DestohovačNaKonecD5 AND ("Dopravník P8 Start" OR (NOT #Přesun.KonecD5naZačátekD8 AND NOT "Paleta na konci P5"))) OR (#Přesun.KonecD5naZačátekD8 AND "Dopravník P8 Start") OR #Přesun.KonecD4naDestohovač))) AND "Silové obvody okruh 1 OK" AND "Motorový jistič P3,P4,P5,P8 OK";
END_REGION

REGION Network 29
   RUNG wire#powerrail
      I_Contact( "Globální řízení_DB".Automat )
      Contact( "OPPovely"."P8 Start" )
      wire#w1
      Coil( "Dopravník P8 Start" )
   END_RUNG
   RUNG wire#powerrail
      Contact( "Globální řízení_DB".Automat )
      wire#w2
      Contact( #Přesun.KonecD5naZačátekD8 )
      wire#w3
      I_Contact( #"Přítomnosti palet".PaletaNaD8pozice12 )
      I_Contact( #Přesun.D8pozice12naD12 )
   END_RUNG wire#w1
   RUNG wire#w3
      Contact( "P12 nahoře" )
   END_RUNG wire#w1
   RUNG wire#w2
      Contact( #Přesun.ZačátekD8naD8pozice12 )
      Contact( "P12 dole" )
   END_RUNG wire#w1
   // the same network as SCL:
   "Dopravník P8 Start" := (NOT "Globální řízení_DB".Automat AND "OPPovely"."P8 Start") OR ("Globální řízení_DB".Automat AND ((#Přesun.KonecD5naZačátekD8 AND ((NOT #"Přítomnosti palet".PaletaNaD8pozice12 AND NOT #Přesun.D8pozice12naD12) OR "P12 nahoře")) OR (#Přesun.ZačátekD8naD8pozice12 AND "P12 dole")));
END_REGION

REGION Network 30
   RUNG wire#powerrail
      I_Contact( "Globální řízení_DB".Automat )
      Contact( "OPPovely"."P12 Nahoru" )
      wire#w1
      I_Contact( "P12 nahoře" )
      I_Contact( "Zdvih P12B Dolu" )
      Coil( "Zdvih P12B Nahoru" )
      wire#w4
      Coil( "Zdvih P12B Brzda" )
   END_RUNG
   RUNG wire#powerrail
      Contact( "Globální řízení_DB".Automat )
      wire#w2
      Contact( #Přesun.D8pozice12naD12 )
      wire#w3
      I_Contact( #Přesun.D17pozice12naKonecP17 )
   END_RUNG wire#w1
   RUNG wire#w2
      Contact( #Přesun.D12naD17pozice12 )
   END_RUNG wire#w3
   RUNG wire#powerrail
      I_Contact( "Globální řízení_DB".Automat )
      Contact( "OPPovely"."P12 Dolu" )
      wire#w5
      I_Contact( "P12 dole" )
      I_Contact( "Zdvih P12B Nahoru" )
      Coil( "Zdvih P12B Dolu" )
   END_RUNG wire#w4
   RUNG wire#powerrail
      Contact( "Globální řízení_DB".Automat )
      wire#w6
      Contact( #Přesun.ZačátekD8naD8pozice12 )
      I_Contact( #Přesun.D12naD17pozice12 )
   END_RUNG wire#w5
   RUNG wire#w6
      Contact( #Přesun.D17pozice12naKonecP17 )
   END_RUNG wire#w5
   RUNG wire#w6
      I_Contact( #Přesun.D8pozice12naD12 )
      I_Contact( #Přesun.D12naD17pozice12 )
   END_RUNG wire#w5
   // the same network as SCL:
   "Zdvih P12B Nahoru" := ((NOT "Globální řízení_DB".Automat AND "OPPovely"."P12 Nahoru") OR ("Globální řízení_DB".Automat AND (#Přesun.D8pozice12naD12 OR #Přesun.D12naD17pozice12) AND NOT #Přesun.D17pozice12naKonecP17)) AND NOT "P12 nahoře" AND NOT "Zdvih P12B Dolu";
   "Zdvih P12B Dolu" := ((NOT "Globální řízení_DB".Automat AND "OPPovely"."P12 Dolu") OR ("Globální řízení_DB".Automat AND ((#Přesun.ZačátekD8naD8pozice12 AND NOT #Přesun.D12naD17pozice12) OR #Přesun.D17pozice12naKonecP17 OR (NOT #Přesun.D8pozice12naD12 AND NOT #Přesun.D12naD17pozice12)))) AND NOT "P12 dole" AND NOT "Zdvih P12B Nahoru";
   "Zdvih P12B Brzda" := "Zdvih P12B Nahoru" OR "Zdvih P12B Dolu";
END_REGION

REGION Network 31
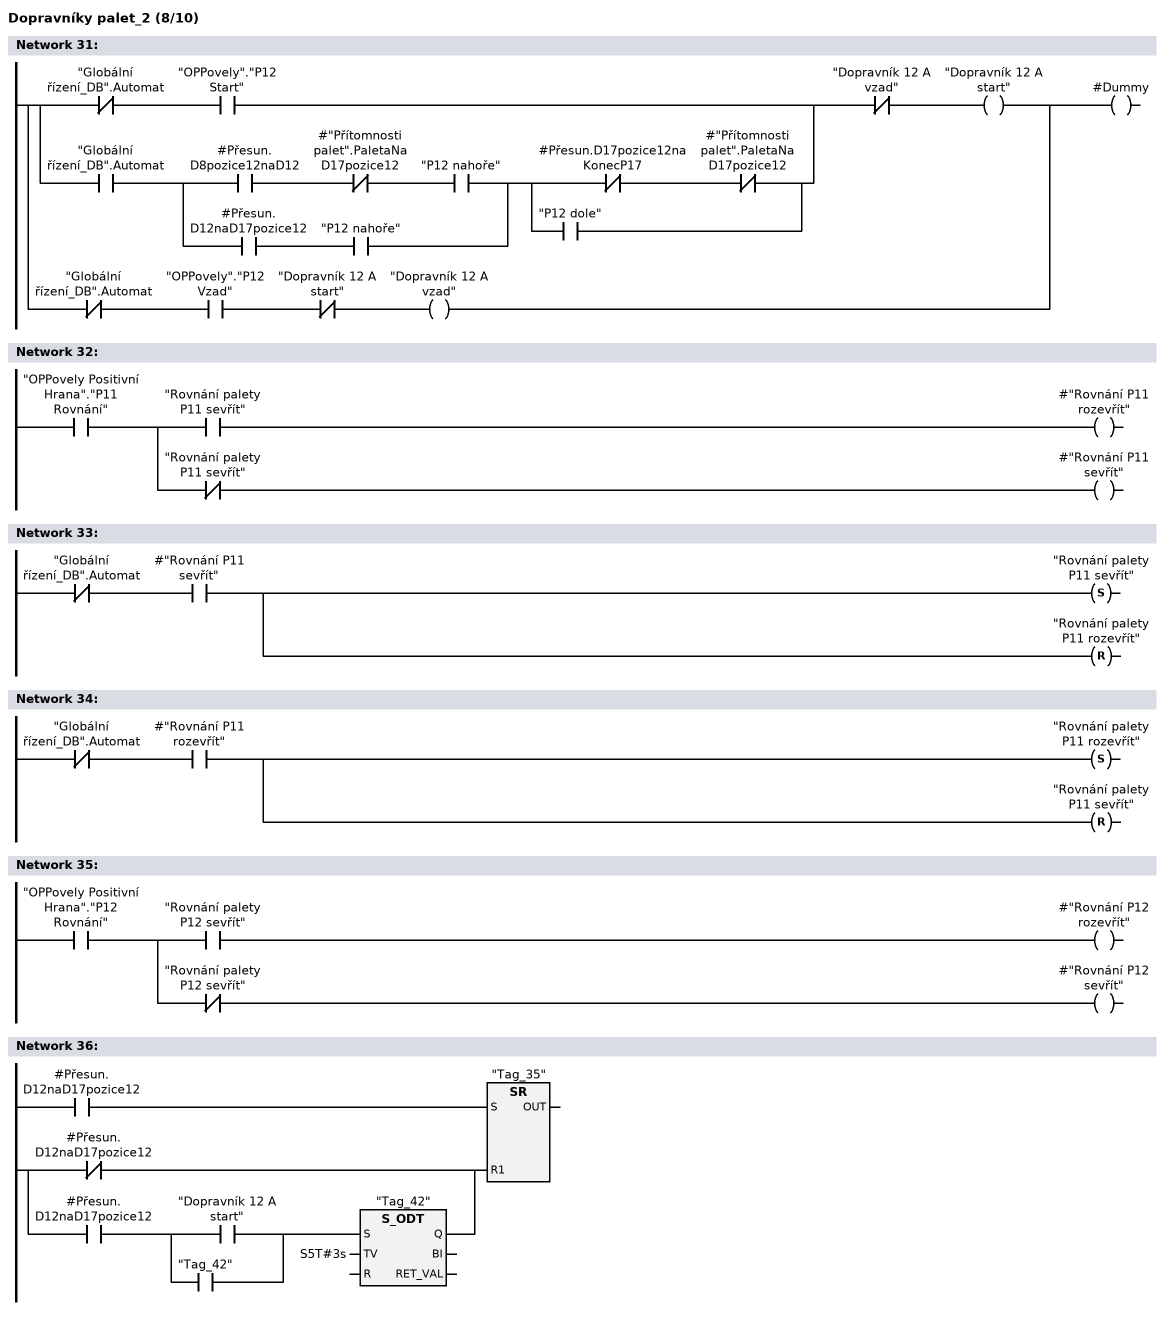
   RUNG wire#powerrail
      I_Contact( "Globální řízení_DB".Automat )
      Contact( "OPPovely"."P12 Start" )
      wire#w1
      I_Contact( "Dopravník 12 A vzad" )
      Coil( "Dopravník 12 A start" )
      wire#w4
      Coil( #Dummy )
   END_RUNG
   RUNG wire#powerrail
      Contact( "Globální řízení_DB".Automat )
      wire#w2
      Contact( #Přesun.D8pozice12naD12 )
      I_Contact( #"Přítomnosti palet".PaletaNaD17pozice12 )
      Contact( "P12 nahoře" )
      wire#w3
      I_Contact( #Přesun.D17pozice12naKonecP17 )
      I_Contact( #"Přítomnosti palet".PaletaNaD17pozice12 )
   END_RUNG wire#w1
   RUNG wire#w2
      Contact( #Přesun.D12naD17pozice12 )
      Contact( "P12 nahoře" )
   END_RUNG wire#w3
   RUNG wire#w3
      Contact( "P12 dole" )
   END_RUNG wire#w1
   RUNG wire#powerrail
      I_Contact( "Globální řízení_DB".Automat )
      Contact( "OPPovely"."P12 Vzad" )
      I_Contact( "Dopravník 12 A start" )
      Coil( "Dopravník 12 A vzad" )
   END_RUNG wire#w4
   // the same network as SCL:
   "Dopravník 12 A start" := ((NOT "Globální řízení_DB".Automat AND "OPPovely"."P12 Start") OR ("Globální řízení_DB".Automat AND ((#Přesun.D8pozice12naD12 AND NOT #"Přítomnosti palet".PaletaNaD17pozice12 AND "P12 nahoře") OR (#Přesun.D12naD17pozice12 AND "P12 nahoře")) AND ((NOT #Přesun.D17pozice12naKonecP17 AND NOT #"Přítomnosti palet".PaletaNaD17pozice12) OR "P12 dole"))) AND NOT "Dopravník 12 A vzad";
   "Dopravník 12 A vzad" := NOT "Globální řízení_DB".Automat AND "OPPovely"."P12 Vzad" AND NOT "Dopravník 12 A start";
   #Dummy := "Dopravník 12 A start" OR "Dopravník 12 A vzad";
END_REGION

REGION Network 32
   RUNG wire#powerrail
      Contact( "OPPovely Positivní Hrana"."P11 Rovnání" )
      wire#w1
      Contact( "Rovnání palety P11 sevřít" )
      Coil( #"Rovnání P11 rozevřít" )
   END_RUNG
   RUNG wire#w1
      I_Contact( "Rovnání palety P11 sevřít" )
      Coil( #"Rovnání P11 sevřít" )
   END_RUNG
   // the same network as SCL:
   #"Rovnání P11 rozevřít" := "OPPovely Positivní Hrana"."P11 Rovnání" AND "Rovnání palety P11 sevřít";
   #"Rovnání P11 sevřít" := "OPPovely Positivní Hrana"."P11 Rovnání" AND NOT "Rovnání palety P11 sevřít";
END_REGION

REGION Network 33
   RUNG wire#powerrail
      I_Contact( "Globální řízení_DB".Automat )
      Contact( #"Rovnání P11 sevřít" )
      wire#w1
      S_Coil( "Rovnání palety P11 sevřít" )
   END_RUNG
   RUNG wire#w1
      R_Coil( "Rovnání palety P11 rozevřít" )
   END_RUNG
   // the same network as SCL:
   IF NOT "Globální řízení_DB".Automat AND #"Rovnání P11 sevřít" THEN
       "Rovnání palety P11 sevřít" := TRUE;
       "Rovnání palety P11 rozevřít" := FALSE;
   END_IF;
END_REGION

REGION Network 34
   RUNG wire#powerrail
      I_Contact( "Globální řízení_DB".Automat )
      Contact( #"Rovnání P11 rozevřít" )
      wire#w1
      S_Coil( "Rovnání palety P11 rozevřít" )
   END_RUNG
   RUNG wire#w1
      R_Coil( "Rovnání palety P11 sevřít" )
   END_RUNG
   // the same network as SCL:
   IF NOT "Globální řízení_DB".Automat AND #"Rovnání P11 rozevřít" THEN
       "Rovnání palety P11 rozevřít" := TRUE;
       "Rovnání palety P11 sevřít" := FALSE;
   END_IF;
END_REGION

REGION Network 35
   RUNG wire#powerrail
      Contact( "OPPovely Positivní Hrana"."P12 Rovnání" )
      wire#w1
      Contact( "Rovnání palety P12 sevřít" )
      Coil( #"Rovnání P12 rozevřít" )
   END_RUNG
   RUNG wire#w1
      I_Contact( "Rovnání palety P12 sevřít" )
      Coil( #"Rovnání P12 sevřít" )
   END_RUNG
   // the same network as SCL:
   #"Rovnání P12 rozevřít" := "OPPovely Positivní Hrana"."P12 Rovnání" AND "Rovnání palety P12 sevřít";
   #"Rovnání P12 sevřít" := "OPPovely Positivní Hrana"."P12 Rovnání" AND NOT "Rovnání palety P12 sevřít";
END_REGION

REGION Network 36
   RUNG wire#powerrail
      Contact( #Přesun.D12naD17pozice12 )
      S_SR(operand := "Tag_35", r1 := wire#w3)
   END_RUNG
   RUNG wire#powerrail
      I_Contact( #Přesun.D12naD17pozice12 )
   END_RUNG wire#w3
   RUNG wire#powerrail
      Contact( #Přesun.D12naD17pozice12 )
      wire#w1
      Contact( "Dopravník 12 A start" )
      wire#w2
      S_ODT(T_NO := "Tag_42", TV := S5T#3s, R :=, BI =>, RET_VAL =>)
   END_RUNG wire#w3
   RUNG wire#w1
      Contact( "Tag_42" )
   END_RUNG wire#w2
   // the same network as SCL:
   #_w2 := #Přesun.D12naD17pozice12;
   #_w3 := NOT #Přesun.D12naD17pozice12;
   #_s5time1 := S_ODT(T_NO := "Tag_42",
                      S := #Přesun.D12naD17pozice12 AND ("Dopravník 12 A start" OR "Tag_42"),
                      TV := S5T#3s,
                      Q => #_w1);
   IF #_w2 THEN
       "Tag_35" := TRUE;   // SR flip-flop
   END_IF;
   IF #_w3 OR #_w1 THEN "Tag_35" := FALSE; END_IF;
END_REGION

REGION Network 37
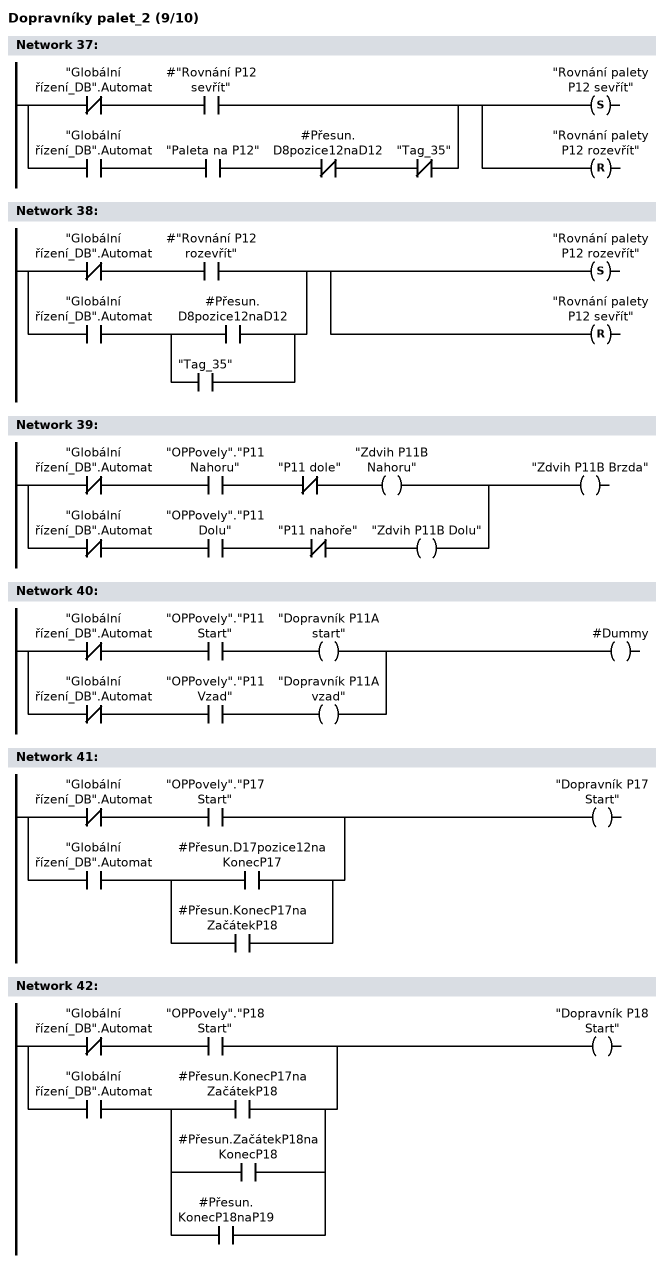
   RUNG wire#powerrail
      I_Contact( "Globální řízení_DB".Automat )
      Contact( #"Rovnání P12 sevřít" )
      wire#w1
      S_Coil( "Rovnání palety P12 sevřít" )
   END_RUNG
   RUNG wire#powerrail
      Contact( "Globální řízení_DB".Automat )
      Contact( "Paleta na P12" )
      I_Contact( #Přesun.D8pozice12naD12 )
      I_Contact( "Tag_35" )
   END_RUNG wire#w1
   RUNG wire#w1
      R_Coil( "Rovnání palety P12 rozevřít" )
   END_RUNG
   // the same network as SCL:
   IF (NOT "Globální řízení_DB".Automat AND #"Rovnání P12 sevřít") OR ("Globální řízení_DB".Automat AND "Paleta na P12" AND NOT #Přesun.D8pozice12naD12 AND NOT "Tag_35") THEN
       "Rovnání palety P12 sevřít" := TRUE;
       "Rovnání palety P12 rozevřít" := FALSE;
   END_IF;
END_REGION

REGION Network 38
   RUNG wire#powerrail
      I_Contact( "Globální řízení_DB".Automat )
      Contact( #"Rovnání P12 rozevřít" )
      wire#w1
      S_Coil( "Rovnání palety P12 rozevřít" )
   END_RUNG
   RUNG wire#powerrail
      Contact( "Globální řízení_DB".Automat )
      wire#w2
      Contact( #Přesun.D8pozice12naD12 )
   END_RUNG wire#w1
   RUNG wire#w2
      Contact( "Tag_35" )
   END_RUNG wire#w1
   RUNG wire#w1
      R_Coil( "Rovnání palety P12 sevřít" )
   END_RUNG
   // the same network as SCL:
   IF (NOT "Globální řízení_DB".Automat AND #"Rovnání P12 rozevřít") OR ("Globální řízení_DB".Automat AND (#Přesun.D8pozice12naD12 OR "Tag_35")) THEN
       "Rovnání palety P12 rozevřít" := TRUE;
       "Rovnání palety P12 sevřít" := FALSE;
   END_IF;
END_REGION

REGION Network 39
   RUNG wire#powerrail
      I_Contact( "Globální řízení_DB".Automat )
      Contact( "OPPovely"."P11 Nahoru" )
      I_Contact( "P11 dole" )
      Coil( "Zdvih P11B Nahoru" )
      wire#w1
      Coil( "Zdvih P11B Brzda" )
   END_RUNG
   RUNG wire#powerrail
      I_Contact( "Globální řízení_DB".Automat )
      Contact( "OPPovely"."P11 Dolu" )
      I_Contact( "P11 nahoře" )
      Coil( "Zdvih P11B Dolu" )
   END_RUNG wire#w1
   // the same network as SCL:
   "Zdvih P11B Nahoru" := NOT "Globální řízení_DB".Automat AND "OPPovely"."P11 Nahoru" AND NOT "P11 dole";
   "Zdvih P11B Dolu" := NOT "Globální řízení_DB".Automat AND "OPPovely"."P11 Dolu" AND NOT "P11 nahoře";
   "Zdvih P11B Brzda" := "Zdvih P11B Nahoru" OR "Zdvih P11B Dolu";
END_REGION

REGION Network 40
   RUNG wire#powerrail
      I_Contact( "Globální řízení_DB".Automat )
      Contact( "OPPovely"."P11 Start" )
      Coil( "Dopravník P11A start" )
      wire#w1
      Coil( #Dummy )
   END_RUNG
   RUNG wire#powerrail
      I_Contact( "Globální řízení_DB".Automat )
      Contact( "OPPovely"."P11 Vzad" )
      Coil( "Dopravník P11A vzad" )
   END_RUNG wire#w1
   // the same network as SCL:
   "Dopravník P11A start" := NOT "Globální řízení_DB".Automat AND "OPPovely"."P11 Start";
   "Dopravník P11A vzad" := NOT "Globální řízení_DB".Automat AND "OPPovely"."P11 Vzad";
   #Dummy := "Dopravník P11A start" OR "Dopravník P11A vzad";
END_REGION

REGION Network 41
   RUNG wire#powerrail
      I_Contact( "Globální řízení_DB".Automat )
      Contact( "OPPovely"."P17 Start" )
      wire#w1
      Coil( "Dopravník P17 Start" )
   END_RUNG
   RUNG wire#powerrail
      Contact( "Globální řízení_DB".Automat )
      wire#w2
      Contact( #Přesun.D17pozice12naKonecP17 )
   END_RUNG wire#w1
   RUNG wire#w2
      Contact( #Přesun.KonecP17naZačátekP18 )
   END_RUNG wire#w1
   // the same network as SCL:
   "Dopravník P17 Start" := (NOT "Globální řízení_DB".Automat AND "OPPovely"."P17 Start") OR ("Globální řízení_DB".Automat AND (#Přesun.D17pozice12naKonecP17 OR #Přesun.KonecP17naZačátekP18));
END_REGION

REGION Network 42
   RUNG wire#powerrail
      I_Contact( "Globální řízení_DB".Automat )
      Contact( "OPPovely"."P18 Start" )
      wire#w1
      Coil( "Dopravník P18 Start" )
   END_RUNG
   RUNG wire#powerrail
      Contact( "Globální řízení_DB".Automat )
      wire#w2
      Contact( #Přesun.KonecP17naZačátekP18 )
   END_RUNG wire#w1
   RUNG wire#w2
      Contact( #Přesun.ZačátekP18naKonecP18 )
   END_RUNG wire#w1
   RUNG wire#w2
      Contact( #Přesun.KonecP18naP19 )
   END_RUNG wire#w1
   // the same network as SCL:
   "Dopravník P18 Start" := (NOT "Globální řízení_DB".Automat AND "OPPovely"."P18 Start") OR ("Globální řízení_DB".Automat AND (#Přesun.KonecP17naZačátekP18 OR #Přesun.ZačátekP18naKonecP18 OR #Přesun.KonecP18naP19));
END_REGION

REGION Network 43
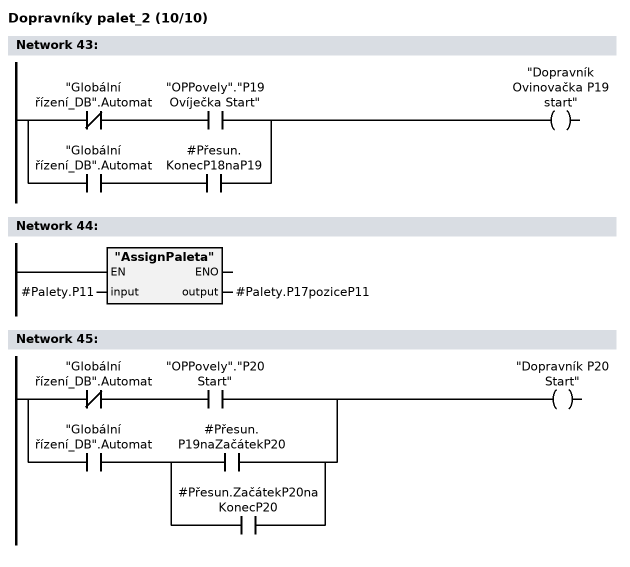
   RUNG wire#powerrail
      I_Contact( "Globální řízení_DB".Automat )
      Contact( "OPPovely"."P19 Ovíječka Start" )
      wire#w1
      Coil( "Dopravník Ovinovačka P19 start" )
   END_RUNG
   RUNG wire#powerrail
      Contact( "Globální řízení_DB".Automat )
      Contact( #Přesun.KonecP18naP19 )
   END_RUNG wire#w1
   // the same network as SCL:
   "Dopravník Ovinovačka P19 start" := (NOT "Globální řízení_DB".Automat AND "OPPovely"."P19 Ovíječka Start") OR ("Globální řízení_DB".Automat AND #Přesun.KonecP18naP19);
END_REGION

REGION Network 44
   RUNG wire#powerrail
      "AssignPaleta"(input := #Palety.P11, output => #Palety.P17poziceP11)
   END_RUNG
   // the same network as SCL:
   "AssignPaleta"(input := #Palety.P11, output => #Palety.P17poziceP11);
END_REGION

REGION Network 45
   RUNG wire#powerrail
      I_Contact( "Globální řízení_DB".Automat )
      Contact( "OPPovely"."P20 Start" )
      wire#w1
      Coil( "Dopravník P20 Start" )
   END_RUNG
   RUNG wire#powerrail
      Contact( "Globální řízení_DB".Automat )
      wire#w2
      Contact( #Přesun.P19naZačátekP20 )
   END_RUNG wire#w1
   RUNG wire#w2
      Contact( #Přesun.ZačátekP20naKonecP20 )
   END_RUNG wire#w1
   // the same network as SCL:
   "Dopravník P20 Start" := (NOT "Globální řízení_DB".Automat AND "OPPovely"."P20 Start") OR ("Globální řízení_DB".Automat AND (#Přesun.P19naZačátekP20 OR #Přesun.ZačátekP20naKonecP20));
END_REGION
END_FUNCTION_BLOCK

FUNCTION_BLOCK "Vyhodnocení hran"   // FB8, LAD
{ S7_Optimized_Access := 'FALSE' }
VERSION : 0.1
   VAR_INPUT
      input : DWord;
   END_VAR
   VAR_OUTPUT
      positive : DInt;
      negative : DInt;
   END_VAR
   VAR
      old_value : DWord;
   END_VAR
   VAR_TEMP
      change : DWord;
      invert : DWord;
   END_VAR
BEGIN

REGION Network 1
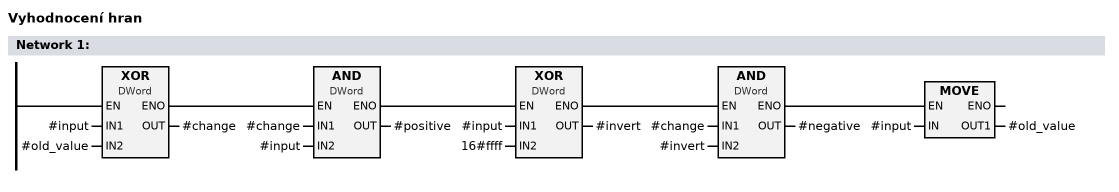
   // no checked SCL form for this network; see the picture
END_REGION
END_FUNCTION_BLOCK

FUNCTION_BLOCK "Přítomnost palety"   // FB9, LAD
{ S7_Optimized_Access := 'FALSE' }
VERSION : 0.1
   VAR_INPUT
      Senzor : Bool;
      Motor : Bool;
      Mezera : S5Time;
      "Reset palety" : Bool;
   END_VAR
   VAR_OUTPUT
      "Nájezd palety" : Bool;
      Paleta : Bool;
   END_VAR
   VAR
      _hrana : Bool;
      _paleta : Bool;
      "_elapsed Time" : DInt;
   END_VAR
   VAR_TEMP
      reset : Bool;
      "time" : Time;
      pv : Time;
      value : DInt;
      te : DInt;
   END_VAR
   VAR_TEMP   // added for the SCL form of the ladder/FBD networks
      _w1 : Bool;
   END_VAR
BEGIN

REGION Network 1
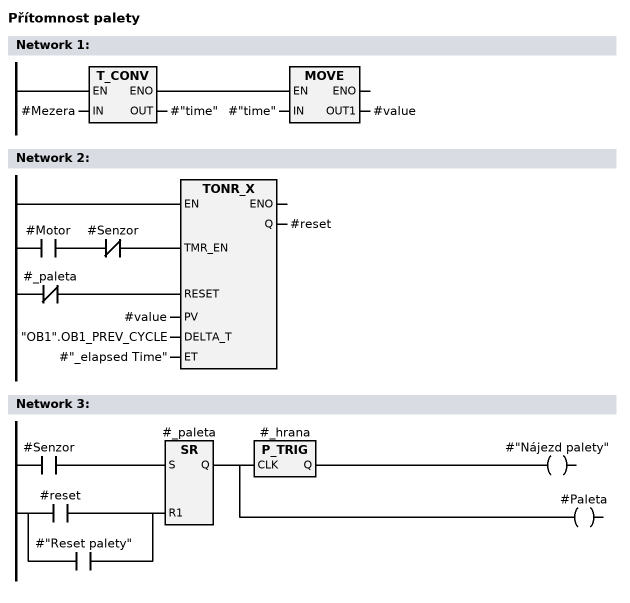
   // ENO of a box is taken as its EN; it also drops when the box reports an error
   #"time" := T_CONV(IN := #Mezera);
   #value := #"time";
END_REGION

REGION Network 2
   TONR_X(TMR_EN := #Motor AND NOT #Senzor,
          RESET := NOT #_paleta,
          PV := #value,
          DELTA_T := "OB1".OB1_PREV_CYCLE,
          ET := #"_elapsed Time",
          Q => #reset);
END_REGION

REGION Network 3
   RUNG wire#powerrail
      Contact( #Senzor )
      S_SR(operand := #_paleta, r1 := wire#w1)
      wire#w2
      P_Trig( #_hrana )
      Coil( #"Nájezd palety" )
   END_RUNG
   RUNG wire#powerrail
      Contact( #reset )
   END_RUNG wire#w1
   RUNG wire#powerrail
      Contact( #"Reset palety" )
   END_RUNG wire#w1
   RUNG wire#w2
      Coil( #Paleta )
   END_RUNG
   // the same network as SCL:
   IF #Senzor THEN
       #_paleta := TRUE;   // SR flip-flop
   END_IF;
   IF #reset OR #"Reset palety" THEN #_paleta := FALSE; END_IF;
   #_w1 := #_paleta AND NOT #_hrana;   // rising edge
   #_hrana := #_paleta;
   #"Nájezd palety" := #_w1;
   #Paleta := #_paleta;
END_REGION
END_FUNCTION_BLOCK

FUNCTION_BLOCK "Dopravníky palet_1"   // FB10, LAD
{ S7_Optimized_Access := 'FALSE' }
VERSION : 0.1
   VAR
      Přesuny : Struct
         PřesunKonecD4naDestohovač : Bool;
         PřesunDestohovačNaKonecD5 : Bool;
         PřesunKonecD5naZačátekD8 : Bool;
         PřesunKonecD8naD8pozice12 : Bool;
         PřesunD8pozice12naD8pozice11 : Bool;
         PřesunD8pozice12naD12 : Bool;
         PřesunD8pozice11naD11 : Bool;
         PřesunD12naD17pozice12 : Bool;
         PřesunD11naD17pozice11 : Bool;
         PřesunD17pozice12naKonecP17 : Bool;
         PřesunD17pozice11naKonecP17 : Bool;
         PřesunKonecP17naZačátekP18 : Bool;
         PřesunZačátekP18naKonecP18 : Bool;
         PřesunKonecP18naP19 : Bool;
         PřesunP19naZačátekP20 : Bool;
         PřesunZačátekP20naKonecP20 : Bool;
         PřesunKonecP20NaP21 : Bool;
      END_STRUCT;
      "Přítomnosti palet" : Struct
         PaletaPodDestohovačem : Bool;
         PaletaNaKonciD5 : Bool;
         PaletaNaZačátkuD8 : Bool;
         PaletaNaD8pozice12 : Bool;
         PaletaNaD8pozice11 : Bool;
         PaletaNaP12 : Bool;
         PaletaNaP11 : Bool;
         PaletaNaD17pozice12 : Bool;
         PaletaNaD17pozice11 : Bool;
         PaletaNaKonciP17 : Bool;
         "PaletaNaZačátku P18" : Bool;
         PaletaNaKonciP18 : Bool;
         PaletaNaP19 : Bool;
         PaletaNaZačátkuP20 : Bool;
         PaletaNaKonciP20 : Bool;
      END_STRUCT;
      "Nájezdy palet" : Struct
         PaletaPodDestohovačem : Bool;
         PaletaNaKonciD5 : Bool;
         PaletaNaZačátkuD8 : Bool;
         PaletaNaD8pozice12 : Bool;
         PaletaNaD8pozice11 : Bool;
         PaletaNaP12 : Bool;
         PaletaNaP11 : Bool;
         PaletaNaD17pozice12 : Bool;
         PaletaNaD17pozice11 : Bool;
         PaletaNaKonciP17 : Bool;
         "PaletaNaZačátku P18" : Bool;
         PaletaNaKonciP18 : Bool;
         PaletaNaP19 : Bool;
         PaletaNaZačátkuP20 : Bool;
         PaletaNaKonciP20 : Bool;
      END_STRUCT;
      Palety : Struct
         P12 : "Paleta";
         P11 : "Paleta";
         P17poziceP11 : "Paleta";
         P17poziceP12 : "Paleta";
         KonecP17 : "Paleta";
         ZačátekP18 : "Paleta";
         KonecP18 : "Paleta";
         P19 : "Paleta";
         ZačátekP20 : "Paleta";
      END_STRUCT;
      Hrany : Struct
         T51Negativní : Bool;
      END_STRUCT;
      "Pallet dispenser_Instance" : "Pallet dispenser";
      "Přítomnost palety_Instance" : "Přítomnost palety";
   END_VAR
   VAR_TEMP
      Dummy : Bool;
      "Rovnání P11 sevřít" : Bool;
      "Rovnání P11 rozevřít" : Bool;
      "Rovnání P12 sevřít" : Bool;
      "Rovnání P12 rozevřít" : Bool;
      "Destohovač sevřít" : Bool;
      "Destohovač rozevřít" : Bool;
   END_VAR
   VAR_TEMP   // added for the SCL form of the ladder/FBD networks
      _s5time1 : S5Time;
   END_VAR
BEGIN

REGION Network 1
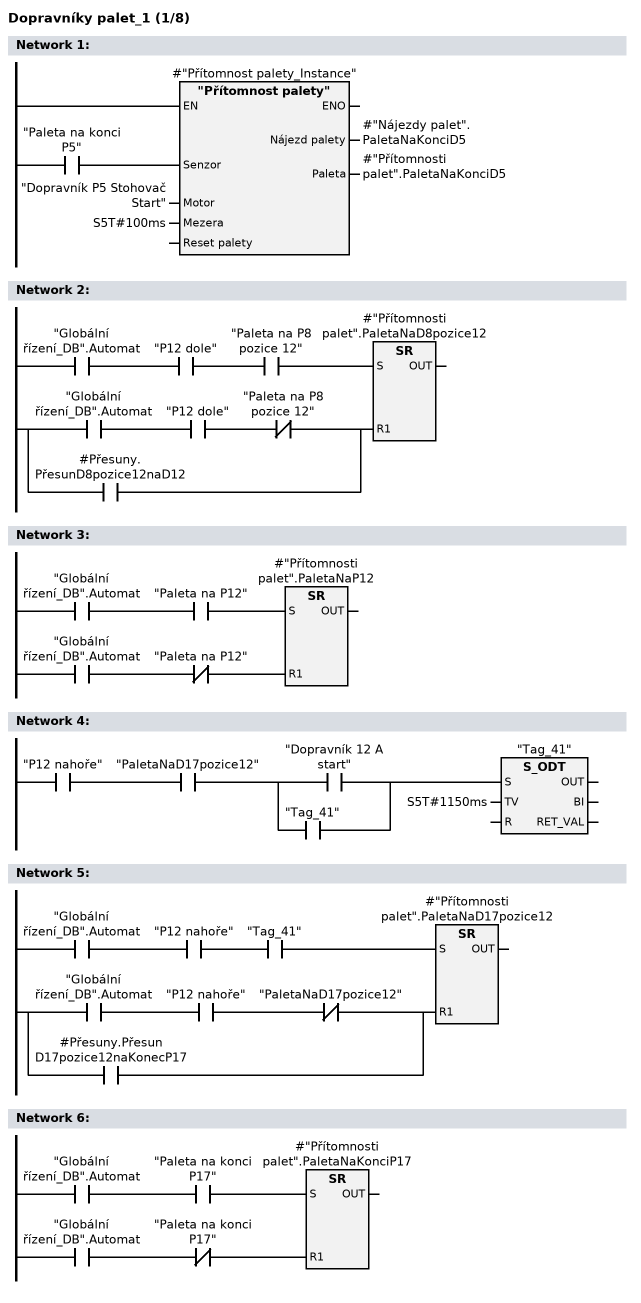
   RUNG wire#powerrail
      #"Přítomnost palety_Instance"(Senzor := wire#w1, Motor := "Dopravník P5 Stohovač Start", Mezera := S5T#100ms, "Reset palety" :=, "Nájezd palety" => #"Nájezdy palet".PaletaNaKonciD5, Paleta => #"Přítomnosti palet".PaletaNaKonciD5)
   END_RUNG
   RUNG wire#powerrail
      Contact( "Paleta na konci P5" )
   END_RUNG wire#w1
   // the same network as SCL:
   #"Přítomnost palety_Instance"(Senzor := "Paleta na konci P5",   // "Přítomnost palety"
                           Motor := "Dopravník P5 Stohovač Start",
                           Mezera := S5T#100ms,
                           "Nájezd palety" => #"Nájezdy palet".PaletaNaKonciD5,
                           Paleta => #"Přítomnosti palet".PaletaNaKonciD5);
END_REGION

REGION Network 2
   RUNG wire#powerrail
      Contact( "Globální řízení_DB".Automat )
      Contact( "P12 dole" )
      Contact( "Paleta na P8 pozice 12" )
      S_SR(operand := #"Přítomnosti palet".PaletaNaD8pozice12, r1 := wire#w1)
   END_RUNG
   RUNG wire#powerrail
      Contact( "Globální řízení_DB".Automat )
      Contact( "P12 dole" )
      I_Contact( "Paleta na P8 pozice 12" )
   END_RUNG wire#w1
   RUNG wire#powerrail
      Contact( #Přesuny.PřesunD8pozice12naD12 )
   END_RUNG wire#w1
   // the same network as SCL:
   IF "Globální řízení_DB".Automat AND "P12 dole" AND "Paleta na P8 pozice 12" THEN
       #"Přítomnosti palet".PaletaNaD8pozice12 := TRUE;   // SR flip-flop
   END_IF;
   IF ("Globální řízení_DB".Automat AND "P12 dole" AND NOT "Paleta na P8 pozice 12") OR #Přesuny.PřesunD8pozice12naD12 THEN
       #"Přítomnosti palet".PaletaNaD8pozice12 := FALSE;
   END_IF;
END_REGION

REGION Network 3
   RUNG wire#powerrail
      Contact( "Globální řízení_DB".Automat )
      Contact( "Paleta na P12" )
      S_SR(operand := #"Přítomnosti palet".PaletaNaP12, r1 := wire#w1)
   END_RUNG
   RUNG wire#powerrail
      Contact( "Globální řízení_DB".Automat )
      I_Contact( "Paleta na P12" )
   END_RUNG wire#w1
   // the same network as SCL:
   IF "Globální řízení_DB".Automat AND "Paleta na P12" THEN
       #"Přítomnosti palet".PaletaNaP12 := TRUE;   // SR flip-flop
   END_IF;
   IF "Globální řízení_DB".Automat AND NOT "Paleta na P12" THEN
       #"Přítomnosti palet".PaletaNaP12 := FALSE;
   END_IF;
END_REGION

REGION Network 4
   RUNG wire#powerrail
      Contact( "P12 nahoře" )
      Contact( "PaletaNaD17pozice12" )
      wire#w1
      Contact( "Dopravník 12 A start" )
      wire#w2
      S_ODT(T_NO := "Tag_41", TV := S5T#1150ms, R :=, BI =>, RET_VAL =>)
   END_RUNG
   RUNG wire#w1
      Contact( "Tag_41" )
   END_RUNG wire#w2
   // the same network as SCL:
   #_s5time1 := S_ODT(T_NO := "Tag_41",
                      S := "P12 nahoře" AND "PaletaNaD17pozice12" AND ("Dopravník 12 A start" OR "Tag_41"),
                      TV := S5T#1150ms);
END_REGION

REGION Network 5
   RUNG wire#powerrail
      Contact( "Globální řízení_DB".Automat )
      Contact( "P12 nahoře" )
      Contact( "Tag_41" )
      S_SR(operand := #"Přítomnosti palet".PaletaNaD17pozice12, r1 := wire#w1)
   END_RUNG
   RUNG wire#powerrail
      Contact( "Globální řízení_DB".Automat )
      Contact( "P12 nahoře" )
      I_Contact( "PaletaNaD17pozice12" )
   END_RUNG wire#w1
   RUNG wire#powerrail
      Contact( #Přesuny.PřesunD17pozice12naKonecP17 )
   END_RUNG wire#w1
   // the same network as SCL:
   IF "Globální řízení_DB".Automat AND "P12 nahoře" AND "Tag_41" THEN
       #"Přítomnosti palet".PaletaNaD17pozice12 := TRUE;   // SR flip-flop
   END_IF;
   IF ("Globální řízení_DB".Automat AND "P12 nahoře" AND NOT "PaletaNaD17pozice12") OR #Přesuny.PřesunD17pozice12naKonecP17 THEN
       #"Přítomnosti palet".PaletaNaD17pozice12 := FALSE;
   END_IF;
END_REGION

REGION Network 6
   RUNG wire#powerrail
      Contact( "Globální řízení_DB".Automat )
      Contact( "Paleta na konci P17" )
      S_SR(operand := #"Přítomnosti palet".PaletaNaKonciP17, r1 := wire#w1)
   END_RUNG
   RUNG wire#powerrail
      Contact( "Globální řízení_DB".Automat )
      I_Contact( "Paleta na konci P17" )
   END_RUNG wire#w1
   // the same network as SCL:
   IF "Globální řízení_DB".Automat AND "Paleta na konci P17" THEN
       #"Přítomnosti palet".PaletaNaKonciP17 := TRUE;   // SR flip-flop
   END_IF;
   IF "Globální řízení_DB".Automat AND NOT "Paleta na konci P17" THEN
       #"Přítomnosti palet".PaletaNaKonciP17 := FALSE;
   END_IF;
END_REGION

REGION Network 7
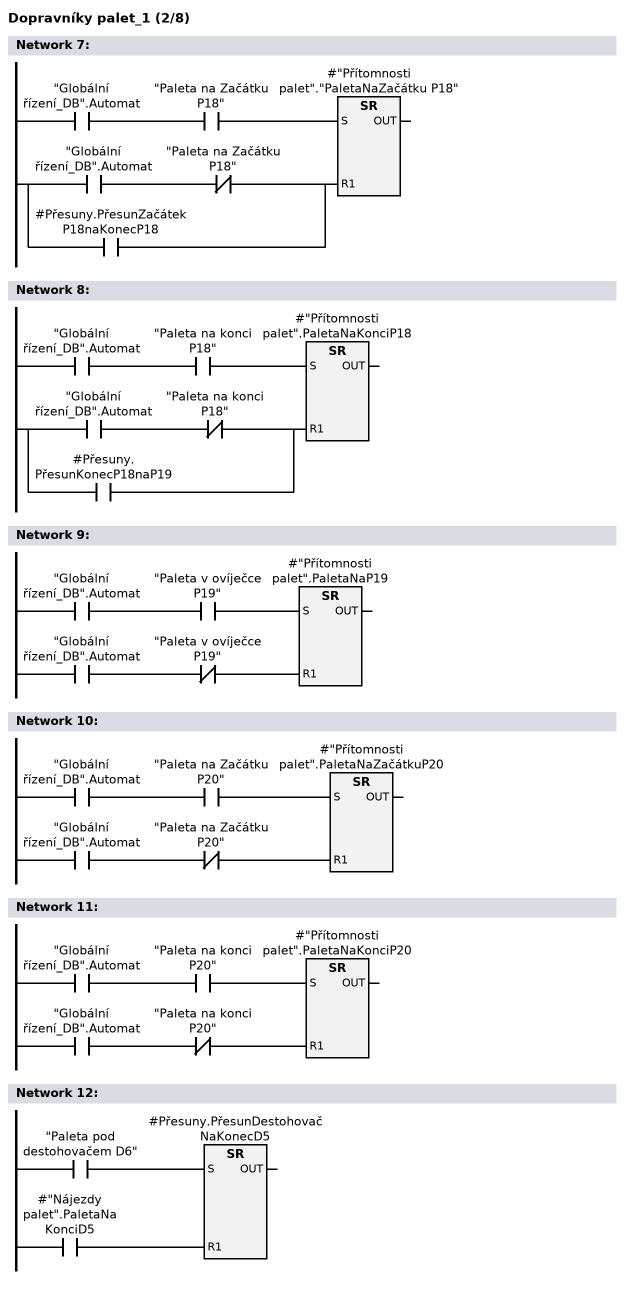
   RUNG wire#powerrail
      Contact( "Globální řízení_DB".Automat )
      Contact( "Paleta na Začátku P18" )
      S_SR(operand := #"Přítomnosti palet"."PaletaNaZačátku P18", r1 := wire#w1)
   END_RUNG
   RUNG wire#powerrail
      Contact( "Globální řízení_DB".Automat )
      I_Contact( "Paleta na Začátku P18" )
   END_RUNG wire#w1
   RUNG wire#powerrail
      Contact( #Přesuny.PřesunZačátekP18naKonecP18 )
   END_RUNG wire#w1
   // the same network as SCL:
   IF "Globální řízení_DB".Automat AND "Paleta na Začátku P18" THEN
       #"Přítomnosti palet"."PaletaNaZačátku P18" := TRUE;   // SR flip-flop
   END_IF;
   IF ("Globální řízení_DB".Automat AND NOT "Paleta na Začátku P18") OR #Přesuny.PřesunZačátekP18naKonecP18 THEN
       #"Přítomnosti palet"."PaletaNaZačátku P18" := FALSE;
   END_IF;
END_REGION

REGION Network 8
   RUNG wire#powerrail
      Contact( "Globální řízení_DB".Automat )
      Contact( "Paleta na konci P18" )
      S_SR(operand := #"Přítomnosti palet".PaletaNaKonciP18, r1 := wire#w1)
   END_RUNG
   RUNG wire#powerrail
      Contact( "Globální řízení_DB".Automat )
      I_Contact( "Paleta na konci P18" )
   END_RUNG wire#w1
   RUNG wire#powerrail
      Contact( #Přesuny.PřesunKonecP18naP19 )
   END_RUNG wire#w1
   // the same network as SCL:
   IF "Globální řízení_DB".Automat AND "Paleta na konci P18" THEN
       #"Přítomnosti palet".PaletaNaKonciP18 := TRUE;   // SR flip-flop
   END_IF;
   IF ("Globální řízení_DB".Automat AND NOT "Paleta na konci P18") OR #Přesuny.PřesunKonecP18naP19 THEN
       #"Přítomnosti palet".PaletaNaKonciP18 := FALSE;
   END_IF;
END_REGION

REGION Network 9
   RUNG wire#powerrail
      Contact( "Globální řízení_DB".Automat )
      Contact( "Paleta v ovíječce P19" )
      S_SR(operand := #"Přítomnosti palet".PaletaNaP19, r1 := wire#w1)
   END_RUNG
   RUNG wire#powerrail
      Contact( "Globální řízení_DB".Automat )
      I_Contact( "Paleta v ovíječce P19" )
   END_RUNG wire#w1
   // the same network as SCL:
   IF "Globální řízení_DB".Automat AND "Paleta v ovíječce P19" THEN
       #"Přítomnosti palet".PaletaNaP19 := TRUE;   // SR flip-flop
   END_IF;
   IF "Globální řízení_DB".Automat AND NOT "Paleta v ovíječce P19" THEN
       #"Přítomnosti palet".PaletaNaP19 := FALSE;
   END_IF;
END_REGION

REGION Network 10
   RUNG wire#powerrail
      Contact( "Globální řízení_DB".Automat )
      Contact( "Paleta na Začátku P20" )
      S_SR(operand := #"Přítomnosti palet".PaletaNaZačátkuP20, r1 := wire#w1)
   END_RUNG
   RUNG wire#powerrail
      Contact( "Globální řízení_DB".Automat )
      I_Contact( "Paleta na Začátku P20" )
   END_RUNG wire#w1
   // the same network as SCL:
   IF "Globální řízení_DB".Automat AND "Paleta na Začátku P20" THEN
       #"Přítomnosti palet".PaletaNaZačátkuP20 := TRUE;   // SR flip-flop
   END_IF;
   IF "Globální řízení_DB".Automat AND NOT "Paleta na Začátku P20" THEN
       #"Přítomnosti palet".PaletaNaZačátkuP20 := FALSE;
   END_IF;
END_REGION

REGION Network 11
   RUNG wire#powerrail
      Contact( "Globální řízení_DB".Automat )
      Contact( "Paleta na konci P20" )
      S_SR(operand := #"Přítomnosti palet".PaletaNaKonciP20, r1 := wire#w1)
   END_RUNG
   RUNG wire#powerrail
      Contact( "Globální řízení_DB".Automat )
      I_Contact( "Paleta na konci P20" )
   END_RUNG wire#w1
   // the same network as SCL:
   IF "Globální řízení_DB".Automat AND "Paleta na konci P20" THEN
       #"Přítomnosti palet".PaletaNaKonciP20 := TRUE;   // SR flip-flop
   END_IF;
   IF "Globální řízení_DB".Automat AND NOT "Paleta na konci P20" THEN
       #"Přítomnosti palet".PaletaNaKonciP20 := FALSE;
   END_IF;
END_REGION

REGION Network 12
   RUNG wire#powerrail
      Contact( "Paleta pod destohovačem D6" )
      S_SR(operand := #Přesuny.PřesunDestohovačNaKonecD5, r1 := wire#w1)
   END_RUNG
   RUNG wire#powerrail
      Contact( #"Nájezdy palet".PaletaNaKonciD5 )
   END_RUNG wire#w1
   // the same network as SCL:
   IF "Paleta pod destohovačem D6" THEN
       #Přesuny.PřesunDestohovačNaKonecD5 := TRUE;   // SR flip-flop
   END_IF;
   IF #"Nájezdy palet".PaletaNaKonciD5 THEN #Přesuny.PřesunDestohovačNaKonecD5 := FALSE; END_IF;
END_REGION

REGION Network 13
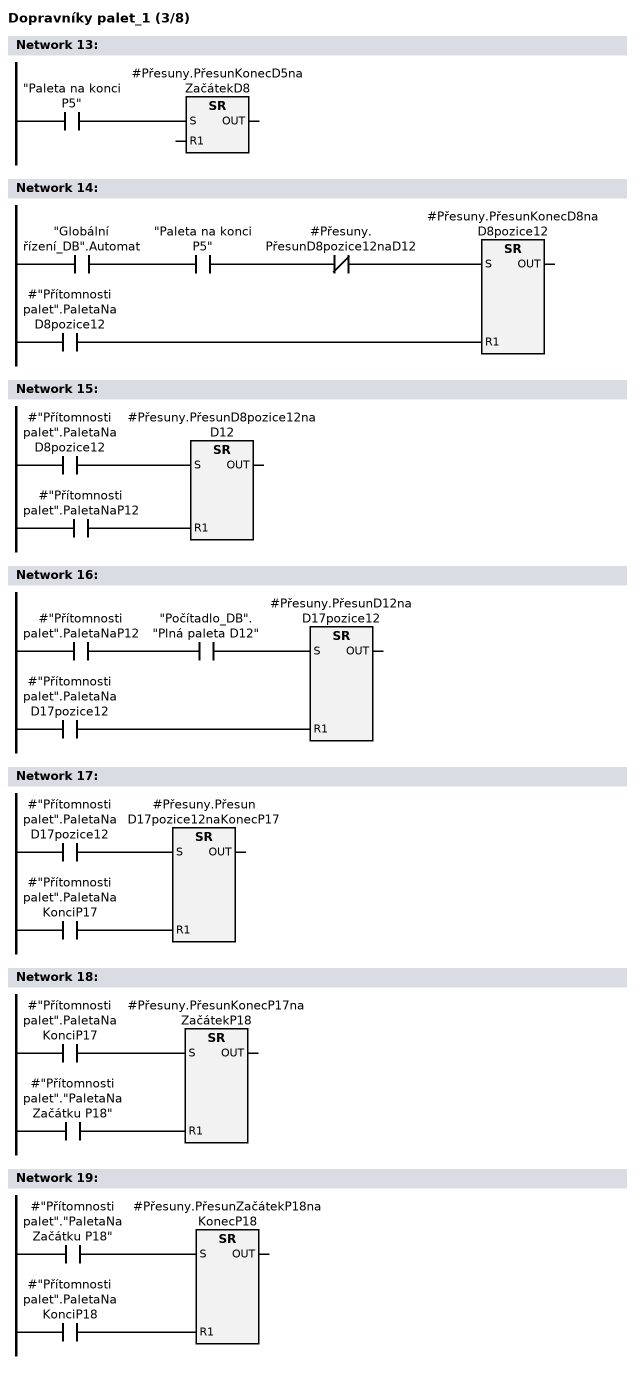
   RUNG wire#powerrail
      Contact( "Paleta na konci P5" )
      S_SR(operand := #Přesuny.PřesunKonecD5naZačátekD8, r1 :=)
   END_RUNG
   // the same network as SCL:
   IF "Paleta na konci P5" THEN
       #Přesuny.PřesunKonecD5naZačátekD8 := TRUE;   // SR flip-flop
   END_IF;
END_REGION

REGION Network 14
   RUNG wire#powerrail
      Contact( "Globální řízení_DB".Automat )
      Contact( "Paleta na konci P5" )
      I_Contact( #Přesuny.PřesunD8pozice12naD12 )
      S_SR(operand := #Přesuny.PřesunKonecD8naD8pozice12, r1 := wire#w1)
   END_RUNG
   RUNG wire#powerrail
      Contact( #"Přítomnosti palet".PaletaNaD8pozice12 )
   END_RUNG wire#w1
   // the same network as SCL:
   IF "Globální řízení_DB".Automat AND "Paleta na konci P5" AND NOT #Přesuny.PřesunD8pozice12naD12 THEN
       #Přesuny.PřesunKonecD8naD8pozice12 := TRUE;   // SR flip-flop
   END_IF;
   IF #"Přítomnosti palet".PaletaNaD8pozice12 THEN #Přesuny.PřesunKonecD8naD8pozice12 := FALSE; END_IF;
END_REGION

REGION Network 15
   RUNG wire#powerrail
      Contact( #"Přítomnosti palet".PaletaNaD8pozice12 )
      S_SR(operand := #Přesuny.PřesunD8pozice12naD12, r1 := wire#w1)
   END_RUNG
   RUNG wire#powerrail
      Contact( #"Přítomnosti palet".PaletaNaP12 )
   END_RUNG wire#w1
   // the same network as SCL:
   IF #"Přítomnosti palet".PaletaNaD8pozice12 THEN
       #Přesuny.PřesunD8pozice12naD12 := TRUE;   // SR flip-flop
   END_IF;
   IF #"Přítomnosti palet".PaletaNaP12 THEN #Přesuny.PřesunD8pozice12naD12 := FALSE; END_IF;
END_REGION

REGION Network 16
   RUNG wire#powerrail
      Contact( #"Přítomnosti palet".PaletaNaP12 )
      Contact( "Počítadlo_DB"."Plná paleta D12" )
      S_SR(operand := #Přesuny.PřesunD12naD17pozice12, r1 := wire#w1)
   END_RUNG
   RUNG wire#powerrail
      Contact( #"Přítomnosti palet".PaletaNaD17pozice12 )
   END_RUNG wire#w1
   // the same network as SCL:
   IF #"Přítomnosti palet".PaletaNaP12 AND "Počítadlo_DB"."Plná paleta D12" THEN
       #Přesuny.PřesunD12naD17pozice12 := TRUE;   // SR flip-flop
   END_IF;
   IF #"Přítomnosti palet".PaletaNaD17pozice12 THEN #Přesuny.PřesunD12naD17pozice12 := FALSE; END_IF;
END_REGION

REGION Network 17
   RUNG wire#powerrail
      Contact( #"Přítomnosti palet".PaletaNaD17pozice12 )
      S_SR(operand := #Přesuny.PřesunD17pozice12naKonecP17, r1 := wire#w1)
   END_RUNG
   RUNG wire#powerrail
      Contact( #"Přítomnosti palet".PaletaNaKonciP17 )
   END_RUNG wire#w1
   // the same network as SCL:
   IF #"Přítomnosti palet".PaletaNaD17pozice12 THEN
       #Přesuny.PřesunD17pozice12naKonecP17 := TRUE;   // SR flip-flop
   END_IF;
   IF #"Přítomnosti palet".PaletaNaKonciP17 THEN #Přesuny.PřesunD17pozice12naKonecP17 := FALSE; END_IF;
END_REGION

REGION Network 18
   RUNG wire#powerrail
      Contact( #"Přítomnosti palet".PaletaNaKonciP17 )
      S_SR(operand := #Přesuny.PřesunKonecP17naZačátekP18, r1 := wire#w1)
   END_RUNG
   RUNG wire#powerrail
      Contact( #"Přítomnosti palet"."PaletaNaZačátku P18" )
   END_RUNG wire#w1
   // the same network as SCL:
   IF #"Přítomnosti palet".PaletaNaKonciP17 THEN
       #Přesuny.PřesunKonecP17naZačátekP18 := TRUE;   // SR flip-flop
   END_IF;
   IF #"Přítomnosti palet"."PaletaNaZačátku P18" THEN #Přesuny.PřesunKonecP17naZačátekP18 := FALSE; END_IF;
END_REGION

REGION Network 19
   RUNG wire#powerrail
      Contact( #"Přítomnosti palet"."PaletaNaZačátku P18" )
      S_SR(operand := #Přesuny.PřesunZačátekP18naKonecP18, r1 := wire#w1)
   END_RUNG
   RUNG wire#powerrail
      Contact( #"Přítomnosti palet".PaletaNaKonciP18 )
   END_RUNG wire#w1
   // the same network as SCL:
   IF #"Přítomnosti palet"."PaletaNaZačátku P18" THEN
       #Přesuny.PřesunZačátekP18naKonecP18 := TRUE;   // SR flip-flop
   END_IF;
   IF #"Přítomnosti palet".PaletaNaKonciP18 THEN #Přesuny.PřesunZačátekP18naKonecP18 := FALSE; END_IF;
END_REGION

REGION Network 20
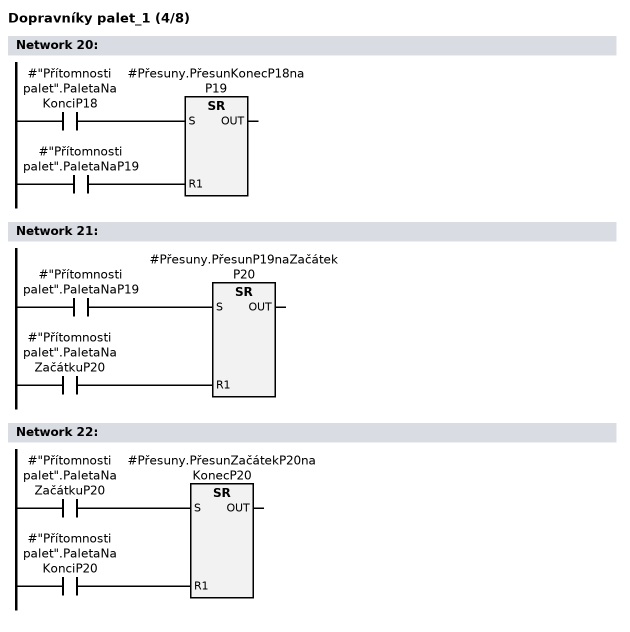
   RUNG wire#powerrail
      Contact( #"Přítomnosti palet".PaletaNaKonciP18 )
      S_SR(operand := #Přesuny.PřesunKonecP18naP19, r1 := wire#w1)
   END_RUNG
   RUNG wire#powerrail
      Contact( #"Přítomnosti palet".PaletaNaP19 )
   END_RUNG wire#w1
   // the same network as SCL:
   IF #"Přítomnosti palet".PaletaNaKonciP18 THEN
       #Přesuny.PřesunKonecP18naP19 := TRUE;   // SR flip-flop
   END_IF;
   IF #"Přítomnosti palet".PaletaNaP19 THEN #Přesuny.PřesunKonecP18naP19 := FALSE; END_IF;
END_REGION

REGION Network 21
   RUNG wire#powerrail
      Contact( #"Přítomnosti palet".PaletaNaP19 )
      S_SR(operand := #Přesuny.PřesunP19naZačátekP20, r1 := wire#w1)
   END_RUNG
   RUNG wire#powerrail
      Contact( #"Přítomnosti palet".PaletaNaZačátkuP20 )
   END_RUNG wire#w1
   // the same network as SCL:
   IF #"Přítomnosti palet".PaletaNaP19 THEN
       #Přesuny.PřesunP19naZačátekP20 := TRUE;   // SR flip-flop
   END_IF;
   IF #"Přítomnosti palet".PaletaNaZačátkuP20 THEN #Přesuny.PřesunP19naZačátekP20 := FALSE; END_IF;
END_REGION

REGION Network 22
   RUNG wire#powerrail
      Contact( #"Přítomnosti palet".PaletaNaZačátkuP20 )
      S_SR(operand := #Přesuny.PřesunZačátekP20naKonecP20, r1 := wire#w1)
   END_RUNG
   RUNG wire#powerrail
      Contact( #"Přítomnosti palet".PaletaNaKonciP20 )
   END_RUNG wire#w1
   // the same network as SCL:
   IF #"Přítomnosti palet".PaletaNaZačátkuP20 THEN
       #Přesuny.PřesunZačátekP20naKonecP20 := TRUE;   // SR flip-flop
   END_IF;
   IF #"Přítomnosti palet".PaletaNaKonciP20 THEN #Přesuny.PřesunZačátekP20naKonecP20 := FALSE; END_IF;
END_REGION

REGION Network 23
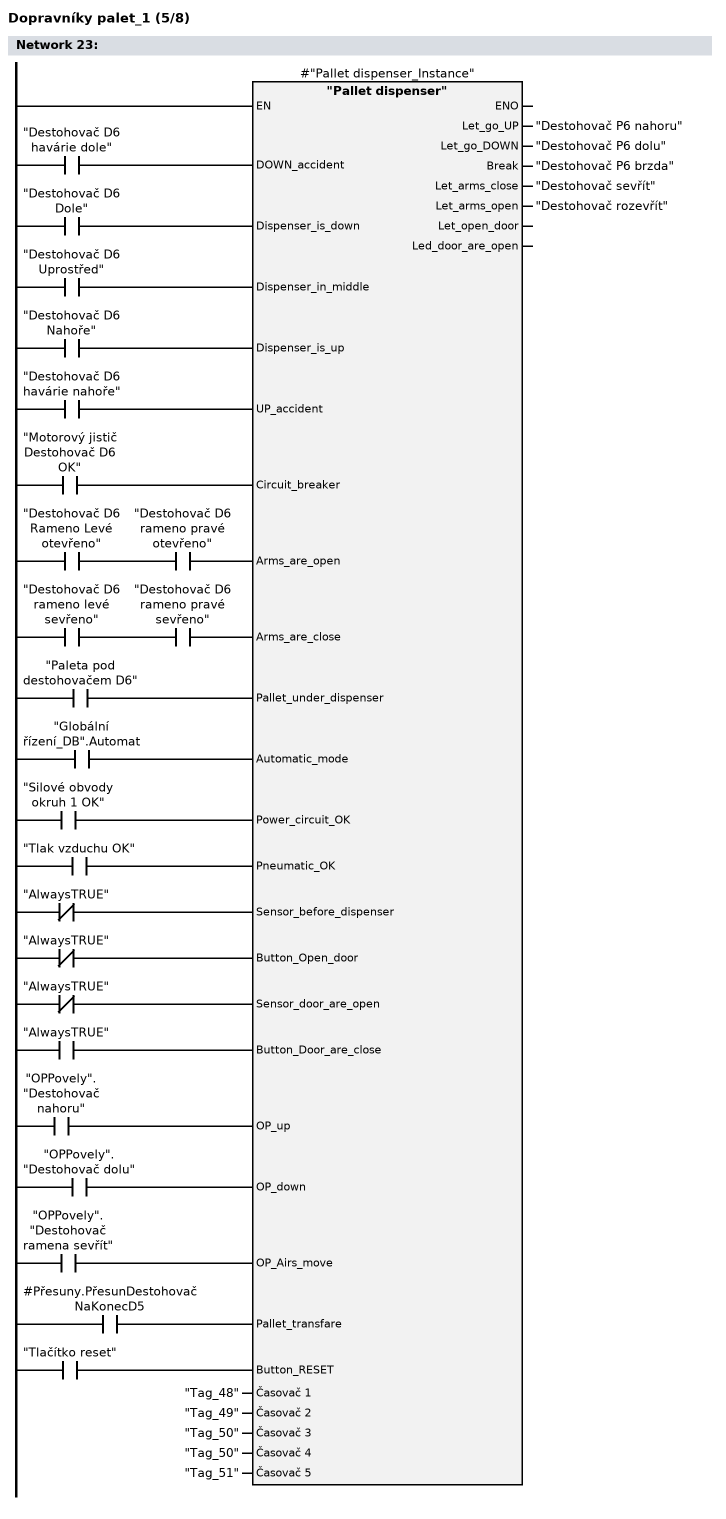
   RUNG wire#powerrail
      #"Pallet dispenser_Instance"(DOWN_accident := wire#w1, Dispenser_is_down := wire#w2, Dispenser_in_middle := wire#w3, Dispenser_is_up := wire#w4, UP_accident := wire#w5, Circuit_breaker := wire#w6, Arms_are_open := wire#w7, Arms_are_close := wire#w8, Pallet_under_dispenser := wire#w9, Automatic_mode := wire#w10, Power_circuit_OK := wire#w11, Pneumatic_OK := wire#w12, Sensor_before_dispenser := wire#w13, Button_Open_door := wire#w14, Sensor_door_are_open := wire#w15, Button_Door_are_close := wire#w16, OP_up := wire#w17, OP_down := wire#w18, OP_Airs_move := wire#w19, Pallet_transfare := wire#w20, Button_RESET := wire#w21, "Časovač 1" := "Tag_48", "Časovač 2" := "Tag_49", "Časovač 3" := "Tag_50", "Časovač 4" := "Tag_50", "Časovač 5" := "Tag_51", Let_go_UP => "Destohovač P6 nahoru", Let_go_DOWN => "Destohovač P6 dolu", Break => "Destohovač P6 brzda", Let_arms_close => "Destohovač sevřít", Let_arms_open => "Destohovač rozevřít", Let_open_door =>, Led_door_are_open =>)
   END_RUNG
   RUNG wire#powerrail
      Contact( "Destohovač D6 havárie dole" )
   END_RUNG wire#w1
   RUNG wire#powerrail
      Contact( "Destohovač D6 Dole" )
   END_RUNG wire#w2
   RUNG wire#powerrail
      Contact( "Destohovač D6 Uprostřed" )
   END_RUNG wire#w3
   RUNG wire#powerrail
      Contact( "Destohovač D6 Nahoře" )
   END_RUNG wire#w4
   RUNG wire#powerrail
      Contact( "Destohovač D6 havárie nahoře" )
   END_RUNG wire#w5
   RUNG wire#powerrail
      Contact( "Motorový jistič Destohovač D6 OK" )
   END_RUNG wire#w6
   RUNG wire#powerrail
      Contact( "Destohovač D6 Rameno Levé otevřeno" )
      Contact( "Destohovač D6 rameno pravé otevřeno" )
   END_RUNG wire#w7
   RUNG wire#powerrail
      Contact( "Destohovač D6 rameno levé sevřeno" )
      Contact( "Destohovač D6 rameno pravé sevřeno" )
   END_RUNG wire#w8
   RUNG wire#powerrail
      Contact( "Paleta pod destohovačem D6" )
   END_RUNG wire#w9
   RUNG wire#powerrail
      Contact( "Globální řízení_DB".Automat )
   END_RUNG wire#w10
   RUNG wire#powerrail
      Contact( "Silové obvody okruh 1 OK" )
   END_RUNG wire#w11
   RUNG wire#powerrail
      Contact( "Tlak vzduchu OK" )
   END_RUNG wire#w12
   RUNG wire#powerrail
      I_Contact( "AlwaysTRUE" )
   END_RUNG wire#w13
   RUNG wire#powerrail
      I_Contact( "AlwaysTRUE" )
   END_RUNG wire#w14
   RUNG wire#powerrail
      I_Contact( "AlwaysTRUE" )
   END_RUNG wire#w15
   RUNG wire#powerrail
      Contact( "AlwaysTRUE" )
   END_RUNG wire#w16
   RUNG wire#powerrail
      Contact( "OPPovely"."Destohovač nahoru" )
   END_RUNG wire#w17
   RUNG wire#powerrail
      Contact( "OPPovely"."Destohovač dolu" )
   END_RUNG wire#w18
   RUNG wire#powerrail
      Contact( "OPPovely"."Destohovač ramena sevřít" )
   END_RUNG wire#w19
   RUNG wire#powerrail
      Contact( #Přesuny.PřesunDestohovačNaKonecD5 )
   END_RUNG wire#w20
   RUNG wire#powerrail
      Contact( "Tlačítko reset" )
   END_RUNG wire#w21
   // the same network as SCL:
   #"Pallet dispenser_Instance"(DOWN_accident := "Destohovač D6 havárie dole",   // "Pallet dispenser"
                           Dispenser_is_down := "Destohovač D6 Dole",
                           Dispenser_in_middle := "Destohovač D6 Uprostřed",
                           Dispenser_is_up := "Destohovač D6 Nahoře",
                           UP_accident := "Destohovač D6 havárie nahoře",
                           Circuit_breaker := "Motorový jistič Destohovač D6 OK",
                           Arms_are_open := "Destohovač D6 Rameno Levé otevřeno" AND "Destohovač D6 rameno pravé otevřeno",
                           Arms_are_close := "Destohovač D6 rameno levé sevřeno" AND "Destohovač D6 rameno pravé sevřeno",
                           Pallet_under_dispenser := "Paleta pod destohovačem D6",
                           Automatic_mode := "Globální řízení_DB".Automat,
                           Power_circuit_OK := "Silové obvody okruh 1 OK",
                           Pneumatic_OK := "Tlak vzduchu OK",
                           Sensor_before_dispenser := NOT "AlwaysTRUE",
                           Button_Open_door := NOT "AlwaysTRUE",
                           Sensor_door_are_open := NOT "AlwaysTRUE",
                           Button_Door_are_close := "AlwaysTRUE",
                           OP_up := "OPPovely"."Destohovač nahoru",
                           OP_down := "OPPovely"."Destohovač dolu",
                           OP_Airs_move := "OPPovely"."Destohovač ramena sevřít",
                           Pallet_transfare := #Přesuny.PřesunDestohovačNaKonecD5,
                           Button_RESET := "Tlačítko reset",
                           "Časovač 1" := "Tag_48",
                           "Časovač 2" := "Tag_49",
                           "Časovač 3" := "Tag_50",
                           "Časovač 4" := "Tag_50",
                           "Časovač 5" := "Tag_51",
                           Let_go_UP => "Destohovač P6 nahoru",
                           Let_go_DOWN => "Destohovač P6 dolu",
                           Break => "Destohovač P6 brzda",
                           Let_arms_close => "Destohovač sevřít",
                           Let_arms_open => "Destohovač rozevřít");
END_REGION

REGION Network 24
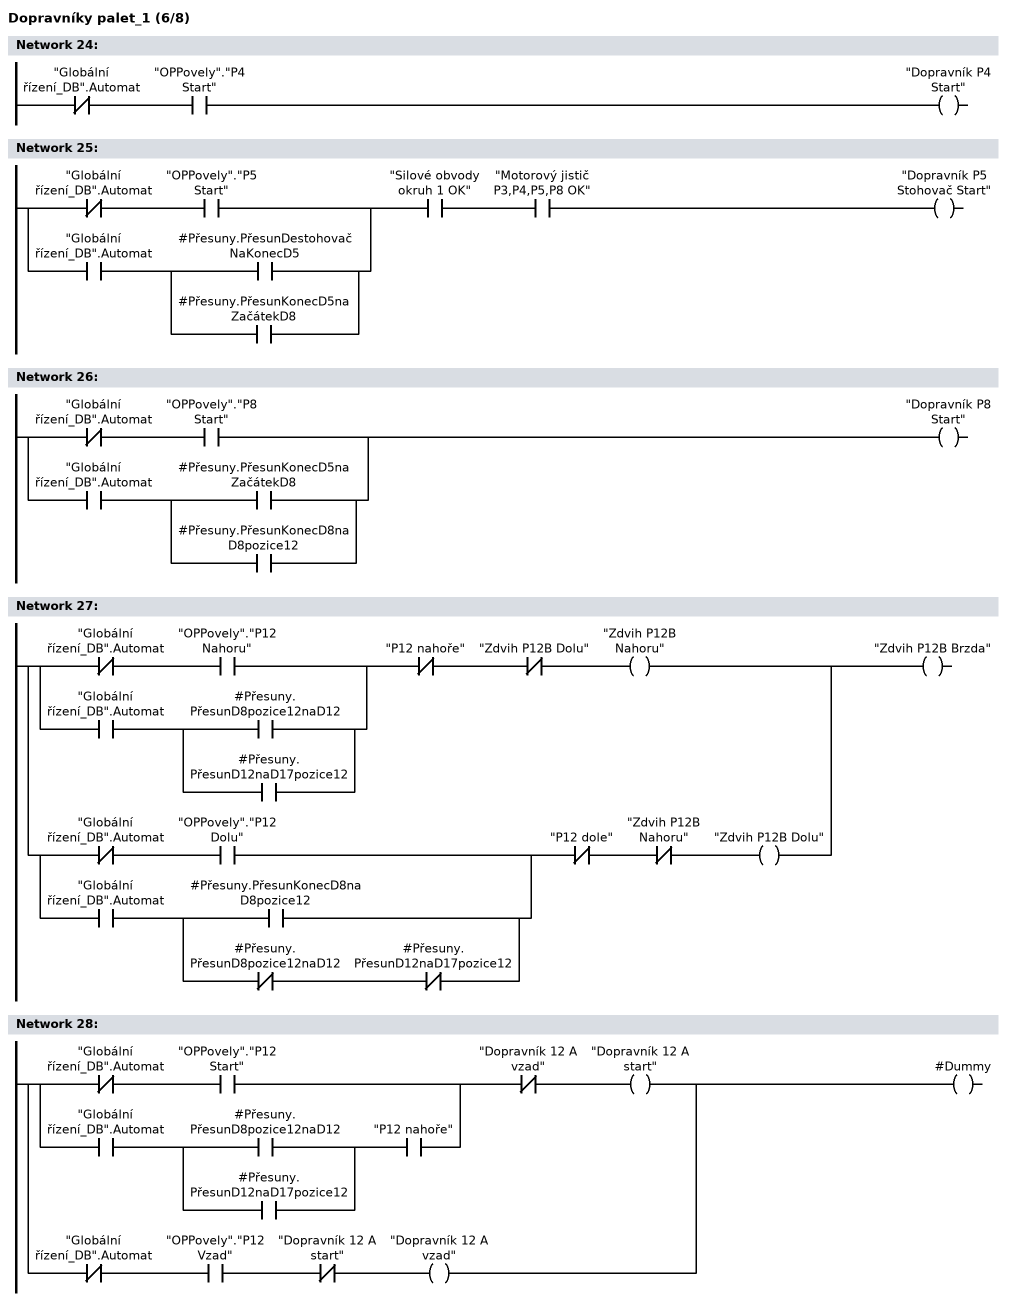
   RUNG wire#powerrail
      I_Contact( "Globální řízení_DB".Automat )
      Contact( "OPPovely"."P4 Start" )
      Coil( "Dopravník P4 Start" )
   END_RUNG
   // the same network as SCL:
   "Dopravník P4 Start" := NOT "Globální řízení_DB".Automat AND "OPPovely"."P4 Start";
END_REGION

REGION Network 25
   RUNG wire#powerrail
      I_Contact( "Globální řízení_DB".Automat )
      Contact( "OPPovely"."P5 Start" )
      wire#w1
      Contact( "Silové obvody okruh 1 OK" )
      Contact( "Motorový jistič P3,P4,P5,P8 OK" )
      Coil( "Dopravník P5 Stohovač Start" )
   END_RUNG
   RUNG wire#powerrail
      Contact( "Globální řízení_DB".Automat )
      wire#w2
      Contact( #Přesuny.PřesunDestohovačNaKonecD5 )
   END_RUNG wire#w1
   RUNG wire#w2
      Contact( #Přesuny.PřesunKonecD5naZačátekD8 )
   END_RUNG wire#w1
   // the same network as SCL:
   "Dopravník P5 Stohovač Start" := ((NOT "Globální řízení_DB".Automat AND "OPPovely"."P5 Start") OR ("Globální řízení_DB".Automat AND (#Přesuny.PřesunDestohovačNaKonecD5 OR #Přesuny.PřesunKonecD5naZačátekD8))) AND "Silové obvody okruh 1 OK" AND "Motorový jistič P3,P4,P5,P8 OK";
END_REGION

REGION Network 26
   RUNG wire#powerrail
      I_Contact( "Globální řízení_DB".Automat )
      Contact( "OPPovely"."P8 Start" )
      wire#w1
      Coil( "Dopravník P8 Start" )
   END_RUNG
   RUNG wire#powerrail
      Contact( "Globální řízení_DB".Automat )
      wire#w2
      Contact( #Přesuny.PřesunKonecD5naZačátekD8 )
   END_RUNG wire#w1
   RUNG wire#w2
      Contact( #Přesuny.PřesunKonecD8naD8pozice12 )
   END_RUNG wire#w1
   // the same network as SCL:
   "Dopravník P8 Start" := (NOT "Globální řízení_DB".Automat AND "OPPovely"."P8 Start") OR ("Globální řízení_DB".Automat AND (#Přesuny.PřesunKonecD5naZačátekD8 OR #Přesuny.PřesunKonecD8naD8pozice12));
END_REGION

REGION Network 27
   RUNG wire#powerrail
      I_Contact( "Globální řízení_DB".Automat )
      Contact( "OPPovely"."P12 Nahoru" )
      wire#w1
      I_Contact( "P12 nahoře" )
      I_Contact( "Zdvih P12B Dolu" )
      Coil( "Zdvih P12B Nahoru" )
      wire#w3
      Coil( "Zdvih P12B Brzda" )
   END_RUNG
   RUNG wire#powerrail
      Contact( "Globální řízení_DB".Automat )
      wire#w2
      Contact( #Přesuny.PřesunD8pozice12naD12 )
   END_RUNG wire#w1
   RUNG wire#w2
      Contact( #Přesuny.PřesunD12naD17pozice12 )
   END_RUNG wire#w1
   RUNG wire#powerrail
      I_Contact( "Globální řízení_DB".Automat )
      Contact( "OPPovely"."P12 Dolu" )
      wire#w4
      I_Contact( "P12 dole" )
      I_Contact( "Zdvih P12B Nahoru" )
      Coil( "Zdvih P12B Dolu" )
   END_RUNG wire#w3
   RUNG wire#powerrail
      Contact( "Globální řízení_DB".Automat )
      wire#w5
      Contact( #Přesuny.PřesunKonecD8naD8pozice12 )
   END_RUNG wire#w4
   RUNG wire#w5
      I_Contact( #Přesuny.PřesunD8pozice12naD12 )
      I_Contact( #Přesuny.PřesunD12naD17pozice12 )
   END_RUNG wire#w4
   // the same network as SCL:
   "Zdvih P12B Nahoru" := ((NOT "Globální řízení_DB".Automat AND "OPPovely"."P12 Nahoru") OR ("Globální řízení_DB".Automat AND (#Přesuny.PřesunD8pozice12naD12 OR #Přesuny.PřesunD12naD17pozice12))) AND NOT "P12 nahoře" AND NOT "Zdvih P12B Dolu";
   "Zdvih P12B Dolu" := ((NOT "Globální řízení_DB".Automat AND "OPPovely"."P12 Dolu") OR ("Globální řízení_DB".Automat AND (#Přesuny.PřesunKonecD8naD8pozice12 OR (NOT #Přesuny.PřesunD8pozice12naD12 AND NOT #Přesuny.PřesunD12naD17pozice12)))) AND NOT "P12 dole" AND NOT "Zdvih P12B Nahoru";
   "Zdvih P12B Brzda" := "Zdvih P12B Nahoru" OR "Zdvih P12B Dolu";
END_REGION

REGION Network 28
   RUNG wire#powerrail
      I_Contact( "Globální řízení_DB".Automat )
      Contact( "OPPovely"."P12 Start" )
      wire#w1
      I_Contact( "Dopravník 12 A vzad" )
      Coil( "Dopravník 12 A start" )
      wire#w4
      Coil( #Dummy )
   END_RUNG
   RUNG wire#powerrail
      Contact( "Globální řízení_DB".Automat )
      wire#w2
      Contact( #Přesuny.PřesunD8pozice12naD12 )
      wire#w3
      Contact( "P12 nahoře" )
   END_RUNG wire#w1
   RUNG wire#w2
      Contact( #Přesuny.PřesunD12naD17pozice12 )
   END_RUNG wire#w3
   RUNG wire#powerrail
      I_Contact( "Globální řízení_DB".Automat )
      Contact( "OPPovely"."P12 Vzad" )
      I_Contact( "Dopravník 12 A start" )
      Coil( "Dopravník 12 A vzad" )
   END_RUNG wire#w4
   // the same network as SCL:
   "Dopravník 12 A start" := ((NOT "Globální řízení_DB".Automat AND "OPPovely"."P12 Start") OR ("Globální řízení_DB".Automat AND (#Přesuny.PřesunD8pozice12naD12 OR #Přesuny.PřesunD12naD17pozice12) AND "P12 nahoře")) AND NOT "Dopravník 12 A vzad";
   "Dopravník 12 A vzad" := NOT "Globální řízení_DB".Automat AND "OPPovely"."P12 Vzad" AND NOT "Dopravník 12 A start";
   #Dummy := "Dopravník 12 A start" OR "Dopravník 12 A vzad";
END_REGION

REGION Network 29
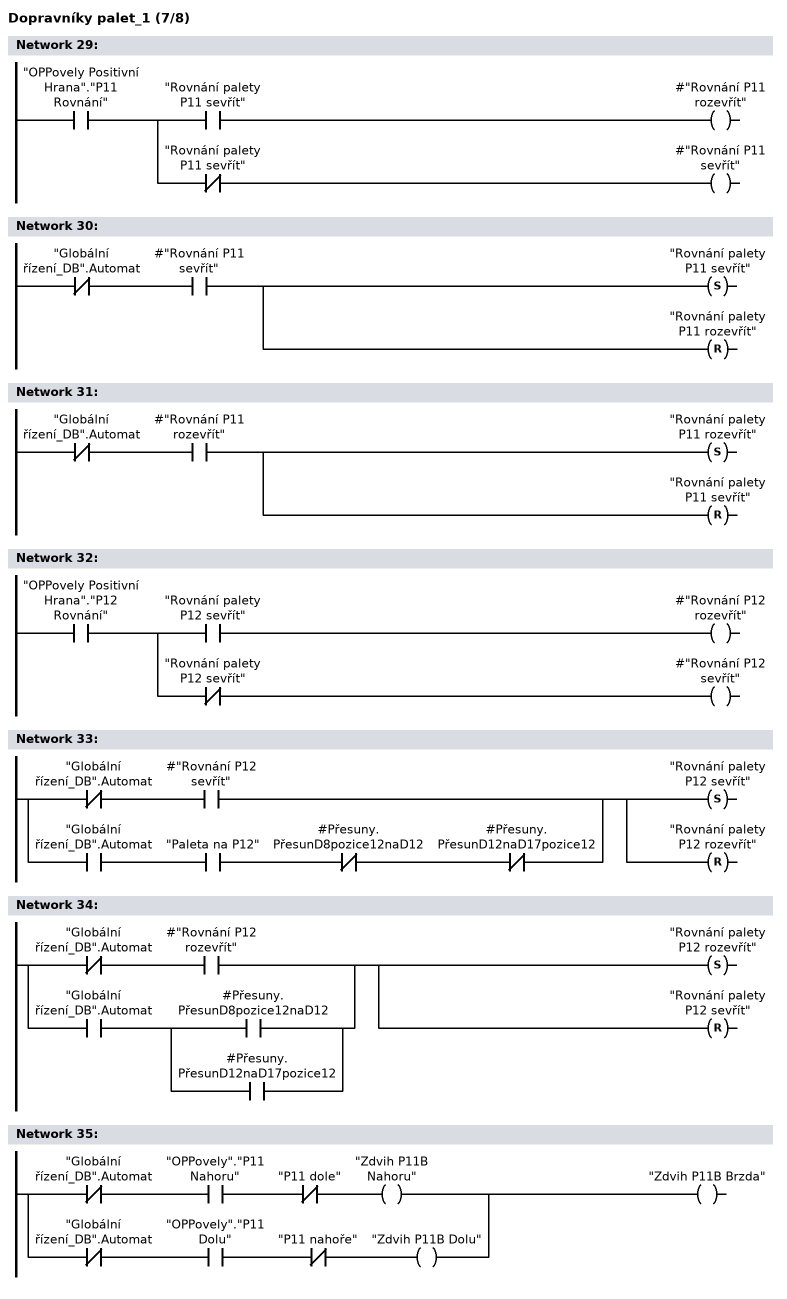
   RUNG wire#powerrail
      Contact( "OPPovely Positivní Hrana"."P11 Rovnání" )
      wire#w1
      Contact( "Rovnání palety P11 sevřít" )
      Coil( #"Rovnání P11 rozevřít" )
   END_RUNG
   RUNG wire#w1
      I_Contact( "Rovnání palety P11 sevřít" )
      Coil( #"Rovnání P11 sevřít" )
   END_RUNG
   // the same network as SCL:
   #"Rovnání P11 rozevřít" := "OPPovely Positivní Hrana"."P11 Rovnání" AND "Rovnání palety P11 sevřít";
   #"Rovnání P11 sevřít" := "OPPovely Positivní Hrana"."P11 Rovnání" AND NOT "Rovnání palety P11 sevřít";
END_REGION

REGION Network 30
   RUNG wire#powerrail
      I_Contact( "Globální řízení_DB".Automat )
      Contact( #"Rovnání P11 sevřít" )
      wire#w1
      S_Coil( "Rovnání palety P11 sevřít" )
   END_RUNG
   RUNG wire#w1
      R_Coil( "Rovnání palety P11 rozevřít" )
   END_RUNG
   // the same network as SCL:
   IF NOT "Globální řízení_DB".Automat AND #"Rovnání P11 sevřít" THEN
       "Rovnání palety P11 sevřít" := TRUE;
       "Rovnání palety P11 rozevřít" := FALSE;
   END_IF;
END_REGION

REGION Network 31
   RUNG wire#powerrail
      I_Contact( "Globální řízení_DB".Automat )
      Contact( #"Rovnání P11 rozevřít" )
      wire#w1
      S_Coil( "Rovnání palety P11 rozevřít" )
   END_RUNG
   RUNG wire#w1
      R_Coil( "Rovnání palety P11 sevřít" )
   END_RUNG
   // the same network as SCL:
   IF NOT "Globální řízení_DB".Automat AND #"Rovnání P11 rozevřít" THEN
       "Rovnání palety P11 rozevřít" := TRUE;
       "Rovnání palety P11 sevřít" := FALSE;
   END_IF;
END_REGION

REGION Network 32
   RUNG wire#powerrail
      Contact( "OPPovely Positivní Hrana"."P12 Rovnání" )
      wire#w1
      Contact( "Rovnání palety P12 sevřít" )
      Coil( #"Rovnání P12 rozevřít" )
   END_RUNG
   RUNG wire#w1
      I_Contact( "Rovnání palety P12 sevřít" )
      Coil( #"Rovnání P12 sevřít" )
   END_RUNG
   // the same network as SCL:
   #"Rovnání P12 rozevřít" := "OPPovely Positivní Hrana"."P12 Rovnání" AND "Rovnání palety P12 sevřít";
   #"Rovnání P12 sevřít" := "OPPovely Positivní Hrana"."P12 Rovnání" AND NOT "Rovnání palety P12 sevřít";
END_REGION

REGION Network 33
   RUNG wire#powerrail
      I_Contact( "Globální řízení_DB".Automat )
      Contact( #"Rovnání P12 sevřít" )
      wire#w1
      S_Coil( "Rovnání palety P12 sevřít" )
   END_RUNG
   RUNG wire#powerrail
      Contact( "Globální řízení_DB".Automat )
      Contact( "Paleta na P12" )
      I_Contact( #Přesuny.PřesunD8pozice12naD12 )
      I_Contact( #Přesuny.PřesunD12naD17pozice12 )
   END_RUNG wire#w1
   RUNG wire#w1
      R_Coil( "Rovnání palety P12 rozevřít" )
   END_RUNG
   // the same network as SCL:
   IF (NOT "Globální řízení_DB".Automat AND #"Rovnání P12 sevřít") OR ("Globální řízení_DB".Automat AND "Paleta na P12" AND NOT #Přesuny.PřesunD8pozice12naD12 AND NOT #Přesuny.PřesunD12naD17pozice12) THEN
       "Rovnání palety P12 sevřít" := TRUE;
       "Rovnání palety P12 rozevřít" := FALSE;
   END_IF;
END_REGION

REGION Network 34
   RUNG wire#powerrail
      I_Contact( "Globální řízení_DB".Automat )
      Contact( #"Rovnání P12 rozevřít" )
      wire#w1
      S_Coil( "Rovnání palety P12 rozevřít" )
   END_RUNG
   RUNG wire#powerrail
      Contact( "Globální řízení_DB".Automat )
      wire#w2
      Contact( #Přesuny.PřesunD8pozice12naD12 )
   END_RUNG wire#w1
   RUNG wire#w2
      Contact( #Přesuny.PřesunD12naD17pozice12 )
   END_RUNG wire#w1
   RUNG wire#w1
      R_Coil( "Rovnání palety P12 sevřít" )
   END_RUNG
   // the same network as SCL:
   IF (NOT "Globální řízení_DB".Automat AND #"Rovnání P12 rozevřít") OR ("Globální řízení_DB".Automat AND (#Přesuny.PřesunD8pozice12naD12 OR #Přesuny.PřesunD12naD17pozice12)) THEN
       "Rovnání palety P12 rozevřít" := TRUE;
       "Rovnání palety P12 sevřít" := FALSE;
   END_IF;
END_REGION

REGION Network 35
   RUNG wire#powerrail
      I_Contact( "Globální řízení_DB".Automat )
      Contact( "OPPovely"."P11 Nahoru" )
      I_Contact( "P11 dole" )
      Coil( "Zdvih P11B Nahoru" )
      wire#w1
      Coil( "Zdvih P11B Brzda" )
   END_RUNG
   RUNG wire#powerrail
      I_Contact( "Globální řízení_DB".Automat )
      Contact( "OPPovely"."P11 Dolu" )
      I_Contact( "P11 nahoře" )
      Coil( "Zdvih P11B Dolu" )
   END_RUNG wire#w1
   // the same network as SCL:
   "Zdvih P11B Nahoru" := NOT "Globální řízení_DB".Automat AND "OPPovely"."P11 Nahoru" AND NOT "P11 dole";
   "Zdvih P11B Dolu" := NOT "Globální řízení_DB".Automat AND "OPPovely"."P11 Dolu" AND NOT "P11 nahoře";
   "Zdvih P11B Brzda" := "Zdvih P11B Nahoru" OR "Zdvih P11B Dolu";
END_REGION

REGION Network 36
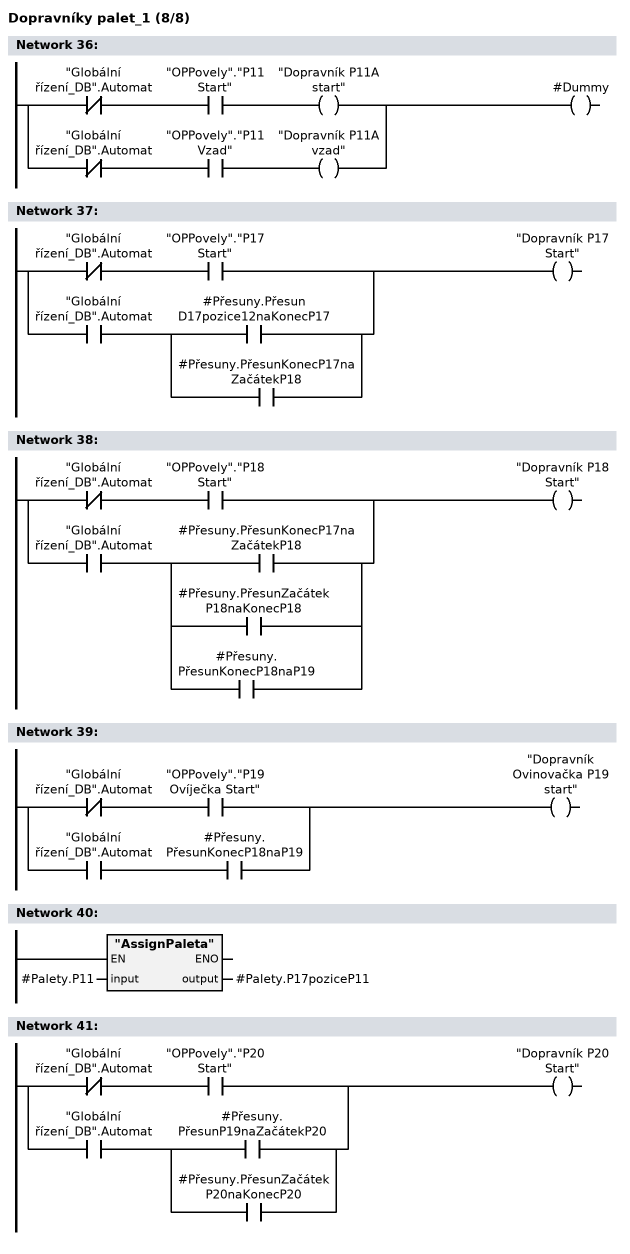
   RUNG wire#powerrail
      I_Contact( "Globální řízení_DB".Automat )
      Contact( "OPPovely"."P11 Start" )
      Coil( "Dopravník P11A start" )
      wire#w1
      Coil( #Dummy )
   END_RUNG
   RUNG wire#powerrail
      I_Contact( "Globální řízení_DB".Automat )
      Contact( "OPPovely"."P11 Vzad" )
      Coil( "Dopravník P11A vzad" )
   END_RUNG wire#w1
   // the same network as SCL:
   "Dopravník P11A start" := NOT "Globální řízení_DB".Automat AND "OPPovely"."P11 Start";
   "Dopravník P11A vzad" := NOT "Globální řízení_DB".Automat AND "OPPovely"."P11 Vzad";
   #Dummy := "Dopravník P11A start" OR "Dopravník P11A vzad";
END_REGION

REGION Network 37
   RUNG wire#powerrail
      I_Contact( "Globální řízení_DB".Automat )
      Contact( "OPPovely"."P17 Start" )
      wire#w1
      Coil( "Dopravník P17 Start" )
   END_RUNG
   RUNG wire#powerrail
      Contact( "Globální řízení_DB".Automat )
      wire#w2
      Contact( #Přesuny.PřesunD17pozice12naKonecP17 )
   END_RUNG wire#w1
   RUNG wire#w2
      Contact( #Přesuny.PřesunKonecP17naZačátekP18 )
   END_RUNG wire#w1
   // the same network as SCL:
   "Dopravník P17 Start" := (NOT "Globální řízení_DB".Automat AND "OPPovely"."P17 Start") OR ("Globální řízení_DB".Automat AND (#Přesuny.PřesunD17pozice12naKonecP17 OR #Přesuny.PřesunKonecP17naZačátekP18));
END_REGION

REGION Network 38
   RUNG wire#powerrail
      I_Contact( "Globální řízení_DB".Automat )
      Contact( "OPPovely"."P18 Start" )
      wire#w1
      Coil( "Dopravník P18 Start" )
   END_RUNG
   RUNG wire#powerrail
      Contact( "Globální řízení_DB".Automat )
      wire#w2
      Contact( #Přesuny.PřesunKonecP17naZačátekP18 )
   END_RUNG wire#w1
   RUNG wire#w2
      Contact( #Přesuny.PřesunZačátekP18naKonecP18 )
   END_RUNG wire#w1
   RUNG wire#w2
      Contact( #Přesuny.PřesunKonecP18naP19 )
   END_RUNG wire#w1
   // the same network as SCL:
   "Dopravník P18 Start" := (NOT "Globální řízení_DB".Automat AND "OPPovely"."P18 Start") OR ("Globální řízení_DB".Automat AND (#Přesuny.PřesunKonecP17naZačátekP18 OR #Přesuny.PřesunZačátekP18naKonecP18 OR #Přesuny.PřesunKonecP18naP19));
END_REGION

REGION Network 39
   RUNG wire#powerrail
      I_Contact( "Globální řízení_DB".Automat )
      Contact( "OPPovely"."P19 Ovíječka Start" )
      wire#w1
      Coil( "Dopravník Ovinovačka P19 start" )
   END_RUNG
   RUNG wire#powerrail
      Contact( "Globální řízení_DB".Automat )
      Contact( #Přesuny.PřesunKonecP18naP19 )
   END_RUNG wire#w1
   // the same network as SCL:
   "Dopravník Ovinovačka P19 start" := (NOT "Globální řízení_DB".Automat AND "OPPovely"."P19 Ovíječka Start") OR ("Globální řízení_DB".Automat AND #Přesuny.PřesunKonecP18naP19);
END_REGION

REGION Network 40
   RUNG wire#powerrail
      "AssignPaleta"(input := #Palety.P11, output => #Palety.P17poziceP11)
   END_RUNG
   // the same network as SCL:
   "AssignPaleta"(input := #Palety.P11, output => #Palety.P17poziceP11);
END_REGION

REGION Network 41
   RUNG wire#powerrail
      I_Contact( "Globální řízení_DB".Automat )
      Contact( "OPPovely"."P20 Start" )
      wire#w1
      Coil( "Dopravník P20 Start" )
   END_RUNG
   RUNG wire#powerrail
      Contact( "Globální řízení_DB".Automat )
      wire#w2
      Contact( #Přesuny.PřesunP19naZačátekP20 )
   END_RUNG wire#w1
   RUNG wire#w2
      Contact( #Přesuny.PřesunZačátekP20naKonecP20 )
   END_RUNG wire#w1
   // the same network as SCL:
   "Dopravník P20 Start" := (NOT "Globální řízení_DB".Automat AND "OPPovely"."P20 Start") OR ("Globální řízení_DB".Automat AND (#Přesuny.PřesunP19naZačátekP20 OR #Přesuny.PřesunZačátekP20naKonecP20));
END_REGION
END_FUNCTION_BLOCK

FUNCTION "AssignPaleta" : Void   // FC1, SCL
{ S7_Optimized_Access := 'FALSE' }
VERSION : 0.1
   VAR_INPUT
      input : "Paleta";
   END_VAR
   VAR_OUTPUT
      output : "Paleta";
   END_VAR
BEGIN
   #output := #input;
END_FUNCTION

FUNCTION "Pulzer" : Void   // FC2, LAD
{ S7_Optimized_Access := 'FALSE' }
VERSION : 0.1
   VAR_INPUT
      T1 : Timer;
      T2 : Timer;
      Thigh : S5Time;
      Tdown : S5Time;
   END_VAR
   VAR_OUTPUT
      Q : Bool;
   END_VAR
   VAR_TEMP   // added for the SCL form of the ladder/FBD networks
      _w1 : Bool;
      _s5time1 : S5Time;
   END_VAR
BEGIN

REGION Network 1
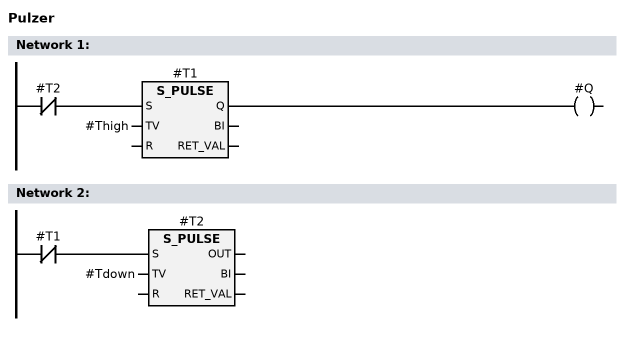
   RUNG wire#powerrail
      I_Contact( #T2 )
      S_PULSE(T_NO := #T1, TV := #Thigh, R :=, BI =>, RET_VAL =>)
      Coil( #Q )
   END_RUNG
   // the same network as SCL:
   #_s5time1 := S_PULSE(T_NO := #T1, S := NOT #T2, TV := #Thigh, Q => #_w1);
   #Q := #_w1;
END_REGION

REGION Network 2
   RUNG wire#powerrail
      I_Contact( #T1 )
      S_PULSE(T_NO := #T2, TV := #Tdown, R :=, BI =>, RET_VAL =>)
   END_RUNG
   // the same network as SCL:
   #_s5time1 := S_PULSE(T_NO := #T2, S := NOT #T1, TV := #Tdown);
END_REGION
END_FUNCTION

ORGANIZATION_BLOCK "Main"   // OB1, LAD
TITLE = "Main Program Sweep (Cycle)"
{ S7_Optimized_Access := 'FALSE' }
VERSION : 0.1
   VAR_TEMP
      OB1_EV_CLASS : Byte;   // Bits 0-3 = 1 (Coming event), Bits 4-7 = 1 (Event class 1)
      OB1_SCAN_1 : Byte;   // 1 (Cold restart scan 1 of OB 1), 3 (Scan 2-n of OB 1)
      OB1_PRIORITY : Byte;   // Priority of OB Execution
      OB1_OB_NUMBR : Byte;   // 1 (Organization block 1, OB1)
      OB1_RESERVED_1 : Byte;   // Reserved for system
      OB1_RESERVED_2 : Byte;   // Reserved for system
      OB1_PREV_CYCLE : Int;   // Cycle time of previous OB1 scan (milliseconds)
      OB1_MIN_CYCLE : Int;   // Minimum cycle time of OB1 (milliseconds)
      OB1_MAX_CYCLE : Int;   // Maximum cycle time of OB1 (milliseconds)
      OB1_DATE_TIME : Date_And_Time;   // Date and time OB1 started
   END_VAR
BEGIN

REGION Network 1
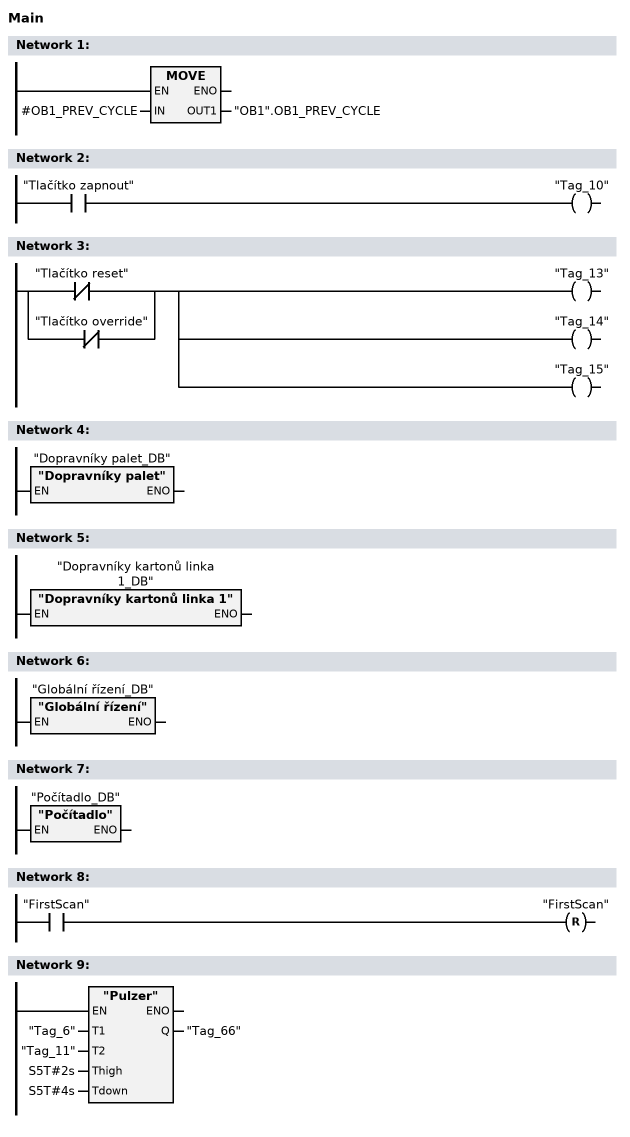
   RUNG wire#powerrail
      { S7_GenerateENO := "TRUE" } Move(in := #OB1_PREV_CYCLE, out1 => "OB1".OB1_PREV_CYCLE)
   END_RUNG
   // the same network as SCL:
   "OB1".OB1_PREV_CYCLE := #OB1_PREV_CYCLE;
END_REGION

REGION Network 2
   RUNG wire#powerrail
      Contact( "Tlačítko zapnout" )
      Coil( "Tag_10" )
   END_RUNG
   // the same network as SCL:
   "Tag_10" := "Tlačítko zapnout";
END_REGION

REGION Network 3
   RUNG wire#powerrail
      I_Contact( "Tlačítko reset" )
      wire#w1
      Coil( "Tag_13" )
   END_RUNG
   RUNG wire#powerrail
      I_Contact( "Tlačítko override" )
   END_RUNG wire#w1
   RUNG wire#w1
      Coil( "Tag_14" )
   END_RUNG
   RUNG wire#w1
      Coil( "Tag_15" )
   END_RUNG
   // the same network as SCL:
   "Tag_13" := NOT "Tlačítko reset" OR NOT "Tlačítko override";
   "Tag_14" := "Tag_13";
   "Tag_15" := "Tag_13";
END_REGION

REGION Network 4
   RUNG wire#powerrail
      "Dopravníky palet_DB"()
   END_RUNG
   // the same network as SCL:
   "Dopravníky palet_DB"();   // "Dopravníky palet"
END_REGION

REGION Network 5
   RUNG wire#powerrail
      "Dopravníky kartonů linka 1_DB"()
   END_RUNG
   // the same network as SCL:
   "Dopravníky kartonů linka 1_DB"();   // "Dopravníky kartonů linka 1"
END_REGION

REGION Network 6
   RUNG wire#powerrail
      "Globální řízení_DB"()
   END_RUNG
   // the same network as SCL:
   "Globální řízení_DB"();   // "Globální řízení"
END_REGION

REGION Network 7
   RUNG wire#powerrail
      "Počítadlo_DB"()
   END_RUNG
   // the same network as SCL:
   "Počítadlo_DB"();   // "Počítadlo"
END_REGION

REGION Network 8
   RUNG wire#powerrail
      Contact( "FirstScan" )
      R_Coil( "FirstScan" )
   END_RUNG
   // the same network as SCL:
   IF "FirstScan" THEN "FirstScan" := FALSE; END_IF;
END_REGION

REGION Network 9
   RUNG wire#powerrail
      "Pulzer"(T1 := "Tag_6", T2 := "Tag_11", Thigh := S5T#2s, Tdown := S5T#4s, Q => "Tag_66")
   END_RUNG
   // the same network as SCL:
   "Pulzer"(T1 := "Tag_6", T2 := "Tag_11", Thigh := S5T#2s, Tdown := S5T#4s, Q => "Tag_66");
END_REGION
END_ORGANIZATION_BLOCK

ORGANIZATION_BLOCK "CYCL_FLT"   // OB80, LAD
TITLE = "Cycle Time Fault"
{ S7_Optimized_Access := 'FALSE' }
VERSION : 0.1
   VAR_TEMP
      OB80_EV_CLASS : Byte;   // 16#35, Event class 3, Entering event state, Internal fault event
      OB80_FLT_ID : Byte;   // 16#XX, Fault identifcation code
      OB80_PRIORITY : Byte;   // Priority of OB Execution
      OB80_OB_NUMBR : Byte;   // 80 (Organization block 80, OB80)
      OB80_RESERVED_1 : Byte;   // Reserved for system
      OB80_RESERVED_2 : Byte;   // Reserved for system
      OB80_ERROR_INFO : Word;   // Error information on event
      OB80_ERR_EV_CLASS : Byte;   // Class of event causing error
      OB80_ERR_EV_NUM : Byte;   // Number of event causing error
      OB80_OB_PRIORITY : Byte;   // Priority of OB causing error
      OB80_OB_NUM : Byte;   // Number of OB causing error
      OB80_DATE_TIME : Date_And_Time;   // Date and time OB80 started
   END_VAR
BEGIN
END_ORGANIZATION_BLOCK

ORGANIZATION_BLOCK "I/O_FLT1"   // OB82, LAD
TITLE = "I/O Point Fault"
{ S7_Optimized_Access := 'FALSE' }
VERSION : 0.1
   VAR_TEMP
      OB82_EV_CLASS : Byte;   // 16#39, Event class 3, Entering event state, Internal fault event
      OB82_FLT_ID : Byte;   // 16#XX, Fault identifcation code
      OB82_PRIORITY : Byte;   // Priority of OB Execution
      OB82_OB_NUMBR : Byte;   // 82 (Organization block 82, OB82)
      OB82_RESERVED_1 : Byte;   // Reserved for system
      OB82_IO_FLAG : Byte;   // Input (01010100), Output (01010101)
      OB82_MDL_ADDR : Word;   // Base address of module with fault
      OB82_MDL_DEFECT : Bool;   // Module defective
      OB82_INT_FAULT : Bool;   // Internal fault
      OB82_EXT_FAULT : Bool;   // External fault
      OB82_PNT_INFO : Bool;   // Point information
      OB82_EXT_VOLTAGE : Bool;   // External voltage low
      OB82_FLD_CONNCTR : Bool;   // Field wiring connector missing
      OB82_NO_CONFIG : Bool;   // Module has no configuration data
      OB82_CONFIG_ERR : Bool;   // Module has configuration error
      OB82_MDL_TYPE : Byte;   // Type of module
      OB82_SUB_MDL_ERR : Bool;   // Sub-Module is missing or has error
      OB82_COMM_FAULT : Bool;   // Communication fault
      OB82_MDL_STOP : Bool;   // Module is stopped
      OB82_WTCH_DOG_FLT : Bool;   // Watch dog timer stopped module
      OB82_INT_PS_FLT : Bool;   // Internal power supply fault
      OB82_PRIM_BATT_FLT : Bool;   // Primary battery is in fault
      OB82_BCKUP_BATT_FLT : Bool;   // Backup battery is in fault
      OB82_RESERVED_2 : Bool;   // Reserved for system
      OB82_RACK_FLT : Bool;   // Rack fault, only for bus interface module
      OB82_PROC_FLT : Bool;   // Processor fault
      OB82_EPROM_FLT : Bool;   // EPROM fault
      OB82_RAM_FLT : Bool;   // RAM fault
      OB82_ADU_FLT : Bool;   // ADU fault
      OB82_FUSE_FLT : Bool;   // Fuse fault
      OB82_HW_INTR_FLT : Bool;   // Hardware interupt input in fault
      OB82_RESERVED_3 : Bool;   // Reserved for system
      OB82_DATE_TIME : Date_And_Time;   // Date and time OB82 started
   END_VAR
BEGIN
END_ORGANIZATION_BLOCK

ORGANIZATION_BLOCK "I/O_FLT2"   // OB83, LAD
TITLE = "I/O Point Fault"
{ S7_Optimized_Access := 'FALSE' }
VERSION : 0.1
   VAR_TEMP
      OB83_EV_CLASS : Byte;   // 16#38/39, Event class 3, module inserted/removed (8/9)
      OB83_FLT_ID : Byte;   // 16#XX, Fault identifcation code
      OB83_PRIORITY : Byte;   // Priority of OB Execution
      OB83_OB_NUMBR : Byte;   // 83 (Organization block 83, OB83)
      OB83_RESERVED_1 : Byte;   // Reserved for system
      OB83_MDL_ID : Byte;   // Input module (01010100), Output module (01010101)
      OB83_MDL_ADDR : Word;   // Base address of module with point fault
      OB83_RACK_NUM : Int;   // Number of rack that has module with point fault
      OB83_MDL_TYPE : Word;   // Module type with point fault
      OB83_DATE_TIME : Date_And_Time;   // Date and time OB83 started
   END_VAR
BEGIN
END_ORGANIZATION_BLOCK

ORGANIZATION_BLOCK "OBNL_FLT"   // OB85, LAD
TITLE = "Organization Block (OB) Not Loaded Fault"
{ S7_Optimized_Access := 'FALSE' }
VERSION : 0.1
   VAR_TEMP
      OB85_EV_CLASS : Byte;   // 16#35 Event class 3
      OB85_FLT_ID : Byte;   // 16#XX, Fault identification code
      OB85_PRIORITY : Byte;   // Priority of OB Execution
      OB85_OB_NUMBR : Byte;   // 85 (Organization block 85, OB85)
      OB85_RESERVED_1 : Byte;   // Reserved for system
      OB85_RESERVED_2 : Byte;   // Reserved for system
      OB85_RESERVED_3 : Int;   // Reserved for system
      OB85_ERR_EV_CLASS : Byte;   // Class of event causing error
      OB85_ERR_EV_NUM : Byte;   // Number of event causing error
      OB85_OB_PRIOR : Byte;   // Priority of OB causing error
      OB85_OB_NUM : Byte;   // Number of OB causing error
      OB85_DATE_TIME : Date_And_Time;   // Date and time OB85 started
   END_VAR
BEGIN
END_ORGANIZATION_BLOCK

ORGANIZATION_BLOCK "RACK_FLT"   // OB86, LAD
TITLE = "Loss Of Rack Fault"
{ S7_Optimized_Access := 'FALSE' }
VERSION : 0.1
   VAR_TEMP
      OB86_EV_CLASS : Byte;   // 16#38/39 Event class 3
      OB86_FLT_ID : Byte;   // 16#C1/C4/C5, Fault identification code
      OB86_PRIORITY : Byte;   // Priority of OB Execution
      OB86_OB_NUMBR : Byte;   // 86 (Organization block 86, OB86)
      OB86_RESERVED_1 : Byte;   // Reserved for system
      OB86_RESERVED_2 : Byte;   // Reserved for system
      OB86_MDL_ADDR : Word;   // Base address of IM module in rack with fault
      OB86_RACKS_FLTD : Array[0..31] of Bool;   // Racks in fault
      OB86_DATE_TIME : Date_And_Time;   // Date and time OB86 started
   END_VAR
BEGIN
END_ORGANIZATION_BLOCK

ORGANIZATION_BLOCK "COMM_FLT"   // OB87, LAD
TITLE = "Communication Fault"
{ S7_Optimized_Access := 'FALSE' }
VERSION : 0.1
   VAR_TEMP
      OB87_EV_CLASS : Byte;   // 16#39 Event class 3
      OB87_FLT_ID : Byte;   // 16#XX, Fault identifcation code
      OB87_PRIORITY : Byte;   // Priority of OB Execution
      OB87_OB_NUMBR : Byte;   // 87 (Organization block 87, OB87)
      OB87_RESERVED_1 : Byte;   // Reserved for system
      OB87_RESERVED_2 : Byte;   // Reserved for system
      OB87_RESERVED_3 : Word;   // Reserved for system
      OB87_RESERVED_4 : DWord;   // Reserved for system
      OB87_DATE_TIME : Date_And_Time;   // Date and time OB87 started
   END_VAR
BEGIN
END_ORGANIZATION_BLOCK

ORGANIZATION_BLOCK "COMPLETE RESTART"   // OB100, LAD
TITLE = "Complete Restart"
{ S7_Optimized_Access := 'FALSE' }
VERSION : 0.1
   VAR_TEMP
      OB100_EV_CLASS : Byte;   // 16#13, Event class 1, Entering event state, Event logged in diagnostic buffer
      OB100_STRTUP : Byte;   // 16#81/82/83/84 Method of startup
      OB100_PRIORITY : Byte;   // Priority of OB Execution
      OB100_OB_NUMBR : Byte;   // 100 (Organization block 100, OB100)
      OB100_RESERVED_1 : Byte;   // Reserved for system
      OB100_RESERVED_2 : Byte;   // Reserved for system
      OB100_STOP : Word;   // Event that caused CPU to stop (16#4xxx)
      OB100_STRT_INFO : DWord;   // Information on how system started
      OB100_DATE_TIME : Date_And_Time;   // Date and time OB100 started
   END_VAR
BEGIN

REGION Network 1
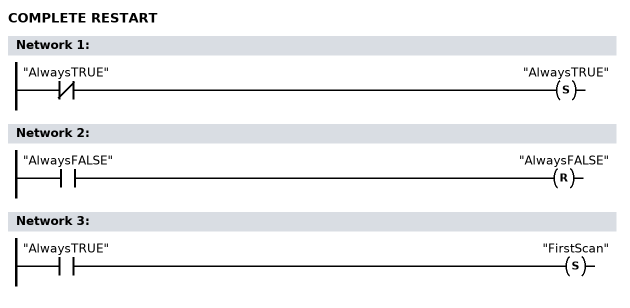
   RUNG wire#powerrail
      I_Contact( "AlwaysTRUE" )
      S_Coil( "AlwaysTRUE" )
   END_RUNG
   // the same network as SCL:
   IF NOT "AlwaysTRUE" THEN "AlwaysTRUE" := TRUE; END_IF;
END_REGION

REGION Network 2
   RUNG wire#powerrail
      Contact( "AlwaysFALSE" )
      R_Coil( "AlwaysFALSE" )
   END_RUNG
   // the same network as SCL:
   IF "AlwaysFALSE" THEN "AlwaysFALSE" := FALSE; END_IF;
END_REGION

REGION Network 3
   RUNG wire#powerrail
      Contact( "AlwaysTRUE" )
      S_Coil( "FirstScan" )
   END_RUNG
   // the same network as SCL:
   IF "AlwaysTRUE" THEN "FirstScan" := TRUE; END_IF;
END_REGION
END_ORGANIZATION_BLOCK

ORGANIZATION_BLOCK "PROG_ERR"   // OB121, LAD
TITLE = "Programming Error"
{ S7_Optimized_Access := 'FALSE' }
VERSION : 0.1
   VAR_TEMP
      OB121_EV_CLASS : Byte;   // 16#25, Event class 2, Entering event state, Internal fault event
      OB121_SW_FLT : Byte;   // 16#XX Software programming fault
      OB121_PRIORITY : Byte;   // Priority of OB Execution
      OB121_OB_NUMBR : Byte;   // 121 (Organization block 121, OB121)
      OB121_BLK_TYPE : Byte;   // 16#88/8A/8B/8C/8E Type of block fault occured in
      OB121_RESERVED_1 : Byte;   // Reserved for system
      OB121_FLT_REG : Word;   // 16#XX Specific register that caused fault
      OB121_BLK_NUM : Word;   // Number of block that programming fault occured in
      OB121_PRG_ADDR : Word;   // Address in block where programming fault occured
      OB121_DATE_TIME : Date_And_Time;   // Date and time OB121 started
   END_VAR
BEGIN
END_ORGANIZATION_BLOCK

ORGANIZATION_BLOCK "MOD_ERR"   // OB122, LAD
TITLE = "Module Access Error"
{ S7_Optimized_Access := 'FALSE' }
VERSION : 0.1
   VAR_TEMP
      OB122_EV_CLASS : Byte;   // 16#29, Event class 2, Entering event state, Internal fault event
      OB122_SW_FLT : Byte;   // 16#XX Software error code
      OB122_PRIORITY : Byte;   // Priority of OB Execution
      OB122_OB_NUMBR : Byte;   // 122 (Organization block 122, OB122)
      OB122_BLK_TYPE : Byte;   // 16#88/8C/8E Type of block fault occured in
      OB122_MEM_AREA : Byte;   // Memory area where access error occured
      OB122_MEM_ADDR : Word;   // Memory address where access error occured
      OB122_BLK_NUM : Word;   // Block number in which error occured
      OB122_PRG_ADDR : Word;   // Program address where error occured
      OB122_DATE_TIME : Date_And_Time;   // Date and time OB1 started
   END_VAR
BEGIN
END_ORGANIZATION_BLOCK

(* ===== HMI "HMI_RT_2" =====
system functions are stored by id; their names below are inferred from use
connection "HMI_Connection_2": ETHERNET, SIMATIC S7 300/400 MPI

